Yaskawa INFORM job: DEMO_ROOF_SIDE_0625_3PAINT_42.JBI

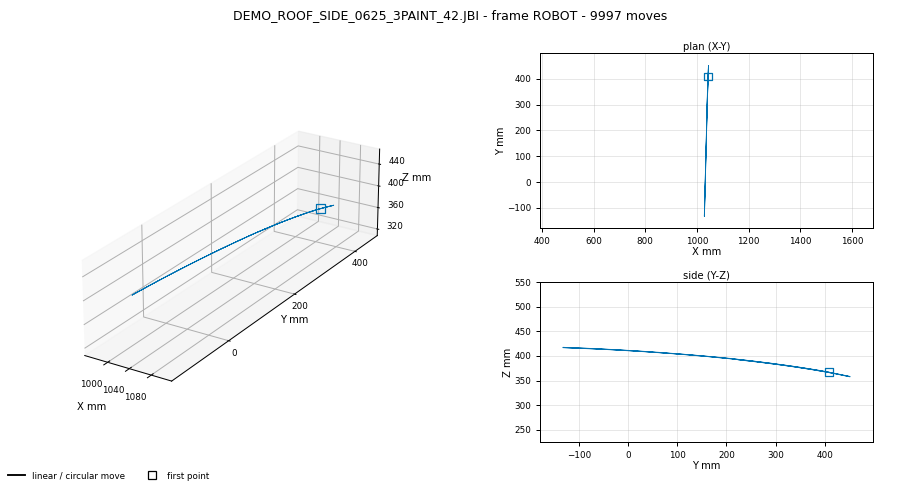
[picture p0: tool path of DEMO_ROOF_SIDE_0625_3PAINT_42.JBI in frame ROBOT, 9997 of 9997 moves have a stored position in this frame; points joined in program order, loops and branches not executed]
/JOB
//NAME DEMO_ROOF_SIDE_0625_3PAINT42
//POS
///NPOS 9997,0,0,0,0,0
///TOOL 0
///USER 0
///POSTYPE ROBOT
///RECTAN
///RCONF 1,0,0,0,0,0,0,0,0,0,0,0,0,0,0,0,0,0,0,0,0,0,0,0
C00000=1043.690,408.820,367.048,174.408,43.868,158.704
C00001=1043.680,408.575,367.094,174.398,43.862,158.701
C00002=1043.671,408.330,367.139,174.389,43.855,158.699
C00003=1043.661,408.085,367.184,174.379,43.848,158.696
C00004=1043.651,407.839,367.230,174.370,43.842,158.694
C00005=1043.642,407.593,367.275,174.361,43.835,158.691
C00006=1043.632,407.347,367.320,174.352,43.829,158.689
C00007=1043.623,407.101,367.365,174.342,43.822,158.686
C00008=1043.613,406.855,367.411,174.333,43.816,158.684
C00009=1043.603,406.610,367.456,174.325,43.809,158.681
C00010=1043.594,406.364,367.501,174.315,43.802,158.679
C00011=1043.586,406.155,367.540,174.308,43.797,158.677
C00012=1043.578,405.946,367.578,174.300,43.791,158.674
C00013=1043.570,405.736,367.616,174.292,43.786,158.672
C00014=1043.561,405.527,367.655,174.284,43.780,158.670
C00015=1043.554,405.317,367.693,174.277,43.775,158.668
C00016=1043.545,405.108,367.732,174.269,43.770,158.666
C00017=1043.537,404.898,367.770,174.261,43.764,158.664
C00018=1043.530,404.689,367.808,174.254,43.759,158.662
C00019=1043.520,404.444,367.853,174.244,43.753,158.660
C00020=1043.511,404.197,367.898,174.235,43.746,158.657
C00021=1043.502,403.952,367.942,174.226,43.740,158.655
C00022=1043.492,403.706,367.987,174.218,43.733,158.652
C00023=1043.483,403.460,368.032,174.209,43.727,158.650
C00024=1043.474,403.214,368.077,174.200,43.721,158.648
C00025=1043.464,402.968,368.121,174.191,43.715,158.645
C00026=1043.454,402.723,368.166,174.183,43.708,158.643
C00027=1043.445,402.477,368.210,174.174,43.702,158.640
C00028=1043.436,402.231,368.255,174.164,43.696,158.638
C00029=1043.427,401.985,368.299,174.156,43.690,158.636
C00030=1043.417,401.740,368.344,174.147,43.684,158.634
C00031=1043.408,401.494,368.388,174.138,43.678,158.631
C00032=1043.399,401.248,368.432,174.130,43.671,158.629
C00033=1043.390,401.002,368.476,174.121,43.666,158.627
C00034=1043.380,400.757,368.521,174.112,43.660,158.624
C00035=1043.371,400.511,368.565,174.104,43.653,158.622
C00036=1043.362,400.264,368.609,174.096,43.648,158.620
C00037=1043.353,400.019,368.653,174.086,43.641,158.617
C00038=1043.344,399.773,368.697,174.079,43.635,158.615
C00039=1043.334,399.527,368.741,174.070,43.630,158.613
C00040=1043.325,399.281,368.785,174.062,43.623,158.611
C00041=1043.315,399.035,368.829,174.053,43.618,158.609
C00042=1043.306,398.789,368.873,174.045,43.612,158.606
C00043=1043.297,398.544,368.917,174.036,43.606,158.604
C00044=1043.288,398.297,368.960,174.028,43.600,158.602
C00045=1043.279,398.051,369.004,174.019,43.594,158.600
C00046=1043.270,397.805,369.048,174.012,43.588,158.598
C00047=1043.261,397.560,369.092,174.003,43.583,158.595
C00048=1043.252,397.313,369.135,173.995,43.577,158.593
C00049=1043.243,397.068,369.179,173.986,43.571,158.591
C00050=1043.234,396.822,369.223,173.978,43.565,158.589
C00051=1043.225,396.575,369.266,173.970,43.559,158.587
C00052=1043.216,396.329,369.310,173.962,43.554,158.584
C00053=1043.206,396.084,369.353,173.953,43.548,158.582
C00054=1043.198,395.838,369.396,173.945,43.542,158.580
C00055=1043.188,395.592,369.440,173.937,43.536,158.578
C00056=1043.180,395.346,369.483,173.929,43.531,158.576
C00057=1043.171,395.100,369.526,173.921,43.525,158.574
C00058=1043.162,394.854,369.570,173.913,43.519,158.572
C00059=1043.153,394.608,369.613,173.905,43.514,158.570
C00060=1043.144,394.362,369.656,173.897,43.508,158.568
C00061=1043.135,394.116,369.700,173.889,43.502,158.565
C00062=1043.126,393.870,369.742,173.880,43.497,158.563
C00063=1043.117,393.624,369.785,173.873,43.491,158.561
C00064=1043.109,393.378,369.828,173.865,43.486,158.559
C00065=1043.100,393.131,369.872,173.856,43.480,158.557
C00066=1043.090,392.886,369.914,173.849,43.475,158.555
C00067=1043.082,392.639,369.957,173.841,43.469,158.553
C00068=1043.073,392.393,370.000,173.833,43.464,158.551
C00069=1043.064,392.148,370.043,173.825,43.458,158.549
C00070=1043.056,391.902,370.086,173.817,43.453,158.547
C00071=1043.041,391.502,370.156,173.805,43.444,158.544
C00072=1043.027,391.102,370.225,173.792,43.435,158.540
C00073=1043.012,390.702,370.294,173.780,43.426,158.537
C00074=1042.998,390.303,370.363,173.767,43.418,158.534
C00075=1042.989,390.057,370.406,173.759,43.413,158.532
C00076=1042.981,389.811,370.449,173.752,43.407,158.530
C00077=1042.972,389.565,370.491,173.744,43.402,158.528
C00078=1042.963,389.319,370.534,173.737,43.397,158.526
C00079=1042.954,389.073,370.576,173.729,43.391,158.524
C00080=1042.946,388.826,370.619,173.722,43.386,158.522
C00081=1042.937,388.580,370.661,173.713,43.381,158.520
C00082=1042.929,388.334,370.703,173.706,43.376,158.519
C00083=1042.919,388.088,370.746,173.698,43.371,158.517
C00084=1042.910,387.842,370.787,173.691,43.365,158.515
C00085=1042.902,387.595,370.830,173.683,43.360,158.513
C00086=1042.893,387.349,370.872,173.676,43.355,158.511
C00087=1042.884,387.103,370.914,173.669,43.350,158.509
C00088=1042.876,386.856,370.956,173.661,43.345,158.507
C00089=1042.867,386.610,370.998,173.654,43.340,158.505
C00090=1042.859,386.364,371.039,173.646,43.334,158.503
C00091=1042.849,386.118,371.082,173.639,43.330,158.502
C00092=1042.841,385.872,371.124,173.632,43.324,158.500
C00093=1042.832,385.625,371.166,173.624,43.319,158.498
C00094=1042.823,385.379,371.207,173.617,43.315,158.496
C00095=1042.815,385.133,371.249,173.609,43.309,158.494
C00096=1042.807,384.887,371.291,173.602,43.304,158.492
C00097=1042.798,384.640,371.333,173.595,43.300,158.490
C00098=1042.789,384.394,371.375,173.588,43.295,158.489
C00099=1042.781,384.148,371.416,173.580,43.289,158.487
C00100=1042.772,383.902,371.458,173.573,43.284,158.485
C00101=1042.763,383.655,371.500,173.566,43.280,158.483
C00102=1042.755,383.409,371.541,173.558,43.275,158.481
C00103=1042.746,383.163,371.582,173.551,43.270,158.480
C00104=1042.738,382.916,371.625,173.545,43.265,158.478
C00105=1042.730,382.670,371.666,173.538,43.260,158.476
C00106=1042.721,382.423,371.707,173.530,43.255,158.474
C00107=1042.712,382.177,371.749,173.523,43.250,158.472
C00108=1042.705,381.931,371.791,173.516,43.245,158.471
C00109=1042.696,381.684,371.832,173.508,43.241,158.469
C00110=1042.688,381.438,371.873,173.501,43.236,158.467
C00111=1042.679,381.192,371.915,173.495,43.231,158.465
C00112=1042.672,380.945,371.956,173.488,43.226,158.464
C00113=1042.663,380.699,371.998,173.480,43.221,158.462
C00114=1042.655,380.453,372.038,173.473,43.217,158.460
C00115=1042.646,380.206,372.080,173.466,43.212,158.458
C00116=1042.638,379.960,372.121,173.460,43.207,158.457
C00117=1042.629,379.713,372.163,173.453,43.202,158.455
C00118=1042.621,379.467,372.203,173.446,43.198,158.453
C00119=1042.613,379.221,372.244,173.438,43.193,158.451
C00120=1042.604,378.974,372.286,173.432,43.188,158.450
C00121=1042.596,378.728,372.326,173.425,43.183,158.448
C00122=1042.588,378.481,372.367,173.418,43.178,158.446
C00123=1042.580,378.235,372.408,173.411,43.174,158.445
C00124=1042.571,377.988,372.449,173.405,43.170,158.443
C00125=1042.563,377.742,372.490,173.398,43.165,158.441
C00126=1042.555,377.495,372.530,173.391,43.160,158.440
C00127=1042.542,377.130,372.591,173.380,43.154,158.437
C00128=1042.530,376.764,372.651,173.370,43.147,158.435
C00129=1042.518,376.398,372.712,173.360,43.140,158.432
C00130=1042.505,376.032,372.772,173.351,43.133,158.430
C00131=1042.497,375.786,372.813,173.344,43.128,158.428
C00132=1042.489,375.539,372.854,173.337,43.124,158.427
C00133=1042.481,375.292,372.894,173.331,43.120,158.425
C00134=1042.472,375.046,372.934,173.324,43.115,158.423
C00135=1042.464,374.799,372.974,173.317,43.111,158.422
C00136=1042.456,374.552,373.015,173.311,43.106,158.420
C00137=1042.448,374.306,373.056,173.304,43.102,158.419
C00138=1042.440,374.059,373.096,173.298,43.098,158.417
C00139=1042.432,373.813,373.137,173.291,43.093,158.416
C00140=1042.424,373.567,373.177,173.284,43.089,158.414
C00141=1042.415,373.319,373.217,173.278,43.084,158.412
C00142=1042.407,373.073,373.257,173.271,43.080,158.411
C00143=1042.399,372.827,373.298,173.265,43.076,158.409
C00144=1042.391,372.580,373.338,173.258,43.071,158.408
C00145=1042.383,372.334,373.379,173.252,43.067,158.406
C00146=1042.375,372.087,373.419,173.245,43.062,158.404
C00147=1042.367,371.840,373.459,173.239,43.058,158.403
C00148=1042.359,371.594,373.499,173.232,43.054,158.401
C00149=1042.351,371.348,373.539,173.226,43.050,158.400
C00150=1042.343,371.101,373.579,173.219,43.045,158.398
C00151=1042.335,370.854,373.619,173.213,43.041,158.397
C00152=1042.327,370.608,373.660,173.206,43.037,158.395
C00153=1042.319,370.361,373.699,173.200,43.032,158.394
C00154=1042.311,370.114,373.739,173.193,43.028,158.392
C00155=1042.303,369.867,373.778,173.188,43.024,158.391
C00156=1042.295,369.621,373.818,173.181,43.020,158.389
C00157=1042.286,369.375,373.858,173.175,43.016,158.388
C00158=1042.278,369.128,373.898,173.169,43.011,158.386
C00159=1042.270,368.881,373.937,173.162,43.007,158.385
C00160=1042.262,368.634,373.977,173.156,43.003,158.383
C00161=1042.254,368.388,374.017,173.149,42.999,158.382
C00162=1042.246,368.141,374.057,173.144,42.995,158.380
C00163=1042.238,367.894,374.096,173.137,42.991,158.379
C00164=1042.230,367.647,374.136,173.131,42.987,158.377
C00165=1042.221,367.401,374.175,173.125,42.983,158.376
C00166=1042.214,367.154,374.215,173.118,42.978,158.374
C00167=1042.206,366.907,374.253,173.112,42.974,158.373
C00168=1042.198,366.660,374.293,173.107,42.970,158.371
C00169=1042.190,366.414,374.333,173.100,42.966,158.370
C00170=1042.182,366.167,374.372,173.094,42.962,158.368
C00171=1042.174,365.920,374.412,173.088,42.958,158.367
C00172=1042.166,365.673,374.452,173.081,42.954,158.366
C00173=1042.158,365.427,374.490,173.076,42.950,158.364
C00174=1042.151,365.180,374.530,173.070,42.946,158.363
C00175=1042.142,364.933,374.569,173.063,42.942,158.361
C00176=1042.135,364.686,374.608,173.057,42.938,158.360
C00177=1042.127,364.440,374.647,173.051,42.934,158.358
C00178=1042.119,364.193,374.687,173.045,42.930,158.357
C00179=1042.111,363.946,374.726,173.039,42.926,158.356
C00180=1042.104,363.699,374.765,173.033,42.922,158.354
C00181=1042.096,363.452,374.804,173.027,42.918,158.353
C00182=1042.088,363.205,374.844,173.021,42.914,158.351
C00183=1042.077,362.859,374.898,173.012,42.909,158.349
C00184=1042.066,362.513,374.953,173.004,42.904,158.348
C00185=1042.056,362.168,375.008,172.997,42.898,158.346
C00186=1042.045,361.821,375.062,172.988,42.893,158.344
C00187=1042.037,361.574,375.101,172.981,42.889,158.342
C00188=1042.028,361.327,375.140,172.976,42.885,158.341
C00189=1042.021,361.081,375.178,172.970,42.881,158.340
C00190=1042.013,360.833,375.218,172.964,42.877,158.338
C00191=1042.006,360.587,375.256,172.959,42.873,158.337
C00192=1041.997,360.340,375.295,172.952,42.870,158.335
C00193=1041.989,360.093,375.334,172.946,42.866,158.334
C00194=1041.982,359.847,375.372,172.941,42.862,158.333
C00195=1041.974,359.599,375.411,172.935,42.859,158.332
C00196=1041.967,359.353,375.450,172.929,42.855,158.330
C00197=1041.959,359.105,375.488,172.923,42.851,158.329
C00198=1041.951,358.859,375.526,172.917,42.847,158.328
C00199=1041.943,358.612,375.565,172.911,42.843,158.326
C00200=1041.935,358.365,375.603,172.906,42.840,158.325
C00201=1041.927,358.118,375.642,172.900,42.836,158.324
C00202=1041.920,357.871,375.680,172.895,42.833,158.322
C00203=1041.912,357.624,375.719,172.889,42.829,158.321
C00204=1041.905,357.377,375.758,172.883,42.825,158.320
C00205=1041.897,357.131,375.796,172.877,42.822,158.318
C00206=1041.889,356.884,375.834,172.871,42.818,158.317
C00207=1041.882,356.636,375.872,172.866,42.814,158.316
C00208=1041.874,356.389,375.911,172.860,42.810,158.314
C00209=1041.866,356.143,375.949,172.854,42.807,158.313
C00210=1041.859,355.896,375.987,172.849,42.803,158.312
C00211=1041.851,355.648,376.025,172.843,42.800,158.311
C00212=1041.843,355.402,376.063,172.838,42.796,158.309
C00213=1041.835,355.155,376.102,172.832,42.793,158.308
C00214=1041.828,354.908,376.139,172.827,42.789,158.307
C00215=1041.820,354.661,376.178,172.821,42.786,158.306
C00216=1041.812,354.413,376.215,172.816,42.782,158.305
C00217=1041.804,354.167,376.253,172.810,42.779,158.303
C00218=1041.797,353.920,376.291,172.804,42.775,158.302
C00219=1041.789,353.673,376.329,172.799,42.771,158.301
C00220=1041.781,353.425,376.367,172.792,42.768,158.299
C00221=1041.774,353.179,376.405,172.787,42.765,158.298
C00222=1041.767,352.932,376.443,172.781,42.761,158.297
C00223=1041.759,352.685,376.481,172.776,42.758,158.296
C00224=1041.751,352.437,376.519,172.771,42.754,158.295
C00225=1041.744,352.191,376.557,172.766,42.751,158.293
C00226=1041.736,351.944,376.594,172.760,42.747,158.292
C00227=1041.729,351.697,376.632,172.755,42.744,158.291
C00228=1041.722,351.450,376.670,172.749,42.740,158.290
C00229=1041.713,351.203,376.707,172.744,42.737,158.288
C00230=1041.706,350.955,376.745,172.738,42.733,158.287
C00231=1041.699,350.708,376.783,172.733,42.730,158.286
C00232=1041.691,350.462,376.821,172.727,42.726,158.285
C00233=1041.684,350.215,376.858,172.722,42.723,158.284
C00234=1041.677,349.968,376.896,172.717,42.720,158.283
C00235=1041.669,349.720,376.933,172.711,42.717,158.281
C00236=1041.661,349.473,376.971,172.706,42.713,158.280
C00237=1041.653,349.226,377.008,172.700,42.710,158.279
C00238=1041.646,348.979,377.046,172.695,42.706,158.278
C00239=1041.636,348.639,377.097,172.688,42.702,158.276
C00240=1041.625,348.299,377.148,172.681,42.697,158.275
C00241=1041.615,347.958,377.200,172.673,42.693,158.273
C00242=1041.604,347.618,377.251,172.666,42.688,158.271
C00243=1041.596,347.371,377.288,172.660,42.685,158.270
C00244=1041.589,347.124,377.326,172.655,42.682,158.269
C00245=1041.582,346.877,377.363,172.650,42.679,158.268
C00246=1041.574,346.630,377.400,172.644,42.675,158.267
C00247=1041.567,346.383,377.438,172.640,42.672,158.266
C00248=1041.560,346.135,377.474,172.634,42.669,158.264
C00249=1041.552,345.888,377.511,172.629,42.666,158.263
C00250=1041.545,345.641,377.549,172.624,42.662,158.262
C00251=1041.537,345.394,377.586,172.618,42.659,158.261
C00252=1041.530,345.146,377.623,172.613,42.656,158.260
C00253=1041.522,344.899,377.660,172.609,42.653,158.259
C00254=1041.515,344.653,377.697,172.603,42.649,158.258
C00255=1041.508,344.405,377.734,172.598,42.646,158.257
C00256=1041.500,344.159,377.771,172.592,42.643,158.255
C00257=1041.493,343.911,377.808,172.587,42.640,158.254
C00258=1041.485,343.664,377.844,172.583,42.637,158.253
C00259=1041.478,343.417,377.882,172.577,42.634,158.252
C00260=1041.471,343.169,377.919,172.572,42.631,158.251
C00261=1041.463,342.922,377.956,172.567,42.628,158.250
C00262=1041.457,342.675,377.992,172.562,42.624,158.249
C00263=1041.449,342.428,378.029,172.557,42.621,158.248
C00264=1041.442,342.181,378.066,172.552,42.618,158.247
C00265=1041.434,341.934,378.103,172.546,42.615,158.245
C00266=1041.427,341.686,378.139,172.542,42.612,158.244
C00267=1041.419,341.439,378.176,172.537,42.609,158.243
C00268=1041.412,341.193,378.212,172.532,42.606,158.242
C00269=1041.404,340.945,378.248,172.526,42.603,158.241
C00270=1041.397,340.697,378.285,172.522,42.599,158.240
C00271=1041.389,340.450,378.322,172.517,42.596,158.239
C00272=1041.381,340.203,378.358,172.511,42.594,158.238
C00273=1041.375,339.956,378.395,172.506,42.591,158.237
C00274=1041.367,339.709,378.431,172.502,42.588,158.236
C00275=1041.360,339.461,378.467,172.496,42.585,158.235
C00276=1041.352,339.214,378.504,172.491,42.582,158.234
C00277=1041.345,338.967,378.541,172.487,42.579,158.233
C00278=1041.338,338.720,378.577,172.482,42.576,158.232
C00279=1041.330,338.472,378.613,172.476,42.573,158.231
C00280=1041.324,338.225,378.650,172.472,42.570,158.230
C00281=1041.316,337.978,378.686,172.467,42.567,158.229
C00282=1041.308,337.730,378.722,172.462,42.564,158.228
C00283=1041.301,337.484,378.758,172.457,42.561,158.227
C00284=1041.294,337.236,378.795,172.452,42.558,158.225
C00285=1041.287,336.988,378.831,172.447,42.555,158.224
C00286=1041.280,336.742,378.867,172.443,42.552,158.223
C00287=1041.272,336.494,378.903,172.437,42.549,158.222
C00288=1041.266,336.247,378.939,172.432,42.546,158.221
C00289=1041.258,336.000,378.976,172.428,42.543,158.220
C00290=1041.250,335.752,379.012,172.423,42.540,158.219
C00291=1041.243,335.506,379.048,172.419,42.538,158.218
C00292=1041.237,335.257,379.084,172.413,42.535,158.217
C00293=1041.230,335.010,379.120,172.408,42.532,158.216
C00294=1041.222,334.763,379.156,172.404,42.529,158.215
C00295=1041.211,334.419,379.205,172.397,42.525,158.214
C00296=1041.201,334.076,379.255,172.390,42.521,158.212
C00297=1041.191,333.732,379.305,172.384,42.517,158.211
C00298=1041.182,333.388,379.355,172.377,42.514,158.210
C00299=1041.174,333.140,379.391,172.372,42.511,158.209
C00300=1041.167,332.893,379.426,172.368,42.507,158.208
C00301=1041.159,332.646,379.463,172.363,42.505,158.207
C00302=1041.153,332.398,379.498,172.357,42.502,158.206
C00303=1041.145,332.151,379.534,172.353,42.499,158.205
C00304=1041.138,331.903,379.569,172.348,42.497,158.204
C00305=1041.131,331.656,379.605,172.344,42.494,158.203
C00306=1041.124,331.409,379.641,172.339,42.491,158.202
C00307=1041.116,331.161,379.677,172.335,42.488,158.201
C00308=1041.109,330.914,379.712,172.329,42.485,158.200
C00309=1041.102,330.667,379.748,172.325,42.483,158.199
C00310=1041.095,330.419,379.783,172.320,42.480,158.198
C00311=1041.088,330.172,379.819,172.316,42.477,158.197
C00312=1041.080,329.924,379.855,172.311,42.474,158.196
C00313=1041.073,329.677,379.890,172.307,42.472,158.195
C00314=1041.067,329.430,379.926,172.302,42.469,158.194
C00315=1041.059,329.182,379.960,172.297,42.467,158.193
C00316=1041.051,328.936,379.996,172.292,42.464,158.192
C00317=1041.045,328.688,380.031,172.288,42.461,158.192
C00318=1041.037,328.440,380.067,172.283,42.459,158.191
C00319=1041.030,328.193,380.101,172.279,42.456,158.190
C00320=1041.022,327.945,380.137,172.274,42.453,158.189
C00321=1041.015,327.698,380.172,172.270,42.451,158.188
C00322=1041.008,327.451,380.207,172.265,42.448,158.187
C00323=1041.000,327.203,380.243,172.261,42.445,158.186
C00324=1040.993,326.956,380.277,172.256,42.443,158.185
C00325=1040.986,326.709,380.313,172.251,42.440,158.184
C00326=1040.978,326.461,380.347,172.246,42.438,158.183
C00327=1040.971,326.214,380.383,172.242,42.435,158.182
C00328=1040.964,325.967,380.417,172.237,42.433,158.181
C00329=1040.956,325.718,380.453,172.233,42.430,158.181
C00330=1040.950,325.471,380.488,172.228,42.428,158.180
C00331=1040.942,325.224,380.522,172.224,42.425,158.179
C00332=1040.935,324.977,380.557,172.219,42.423,158.178
C00333=1040.928,324.728,380.592,172.215,42.420,158.177
C00334=1040.921,324.481,380.627,172.211,42.417,158.176
C00335=1040.913,324.234,380.661,172.206,42.415,158.175
C00336=1040.907,323.987,380.696,172.202,42.412,158.174
C00337=1040.898,323.739,380.731,172.197,42.410,158.173
C00338=1040.892,323.491,380.766,172.193,42.408,158.173
C00339=1040.885,323.244,380.802,172.188,42.405,158.172
C00340=1040.878,322.996,380.835,172.184,42.403,158.171
C00341=1040.871,322.749,380.871,172.180,42.400,158.170
C00342=1040.863,322.502,380.905,172.174,42.398,158.169
C00343=1040.856,322.254,380.941,172.170,42.395,158.168
C00344=1040.849,322.006,380.974,172.166,42.392,158.167
C00345=1040.842,321.759,381.010,172.161,42.390,158.166
C00346=1040.835,321.512,381.044,172.157,42.387,158.166
C00347=1040.828,321.264,381.079,172.152,42.385,158.165
C00348=1040.821,321.017,381.113,172.148,42.382,158.164
C00349=1040.814,320.769,381.148,172.144,42.380,158.163
C00350=1040.807,320.522,381.182,172.139,42.377,158.162
C00351=1040.797,320.173,381.232,172.134,42.374,158.161
C00352=1040.787,319.825,381.280,172.127,42.370,158.160
C00353=1040.777,319.476,381.329,172.121,42.367,158.158
C00354=1040.767,319.127,381.377,172.115,42.363,158.157
C00355=1040.760,318.879,381.412,172.110,42.362,158.156
C00356=1040.753,318.632,381.446,172.106,42.359,158.156
C00357=1040.746,318.384,381.481,172.102,42.357,158.155
C00358=1040.739,318.137,381.515,172.097,42.354,158.154
C00359=1040.732,317.889,381.550,172.093,42.352,158.153
C00360=1040.725,317.642,381.584,172.089,42.349,158.152
C00361=1040.718,317.394,381.619,172.085,42.347,158.151
C00362=1040.711,317.147,381.653,172.080,42.344,158.150
C00363=1040.704,316.899,381.688,172.076,42.342,158.150
C00364=1040.697,316.651,381.721,172.072,42.340,158.149
C00365=1040.691,316.405,381.756,172.068,42.337,158.148
C00366=1040.684,316.157,381.790,172.063,42.335,158.147
C00367=1040.677,315.909,381.824,172.059,42.332,158.146
C00368=1040.670,315.662,381.859,172.055,42.330,158.145
C00369=1040.663,315.414,381.893,172.052,42.328,158.145
C00370=1040.656,315.166,381.927,172.046,42.326,158.144
C00371=1040.649,314.919,381.962,172.042,42.323,158.143
C00372=1040.643,314.672,381.996,172.038,42.320,158.142
C00373=1040.636,314.424,382.030,172.034,42.318,158.141
C00374=1040.629,314.176,382.064,172.030,42.316,158.141
C00375=1040.622,313.929,382.099,172.026,42.314,158.140
C00376=1040.615,313.681,382.133,172.022,42.311,158.139
C00377=1040.609,313.434,382.167,172.018,42.309,158.138
C00378=1040.601,313.187,382.200,172.014,42.307,158.137
C00379=1040.595,312.939,382.235,172.010,42.304,158.137
C00380=1040.588,312.691,382.269,172.005,42.302,158.136
C00381=1040.582,312.444,382.303,172.001,42.300,158.135
C00382=1040.574,312.197,382.337,171.997,42.297,158.134
C00383=1040.567,311.949,382.371,171.993,42.295,158.133
C00384=1040.560,311.701,382.404,171.989,42.293,158.133
C00385=1040.553,311.453,382.438,171.984,42.290,158.132
C00386=1040.547,311.206,382.471,171.980,42.288,158.131
C00387=1040.539,310.958,382.505,171.976,42.286,158.130
C00388=1040.532,310.711,382.539,171.972,42.284,158.129
C00389=1040.524,310.463,382.572,171.968,42.282,158.129
C00390=1040.517,310.216,382.606,171.963,42.280,158.128
C00391=1040.511,309.968,382.639,171.960,42.278,158.127
C00392=1040.504,309.720,382.673,171.956,42.276,158.126
C00393=1040.496,309.473,382.706,171.952,42.273,158.126
C00394=1040.489,309.225,382.740,171.947,42.271,158.125
C00395=1040.483,308.978,382.773,171.943,42.269,158.124
C00396=1040.476,308.730,382.807,171.939,42.267,158.123
C00397=1040.468,308.482,382.840,171.935,42.265,158.123
C00398=1040.460,308.235,382.874,171.931,42.262,158.122
C00399=1040.454,307.987,382.907,171.928,42.260,158.121
C00400=1040.447,307.740,382.940,171.923,42.259,158.120
C00401=1040.440,307.491,382.974,171.919,42.256,158.120
C00402=1040.433,307.244,383.007,171.915,42.254,158.119
C00403=1040.426,306.997,383.040,171.911,42.252,158.118
C00404=1040.419,306.749,383.073,171.907,42.250,158.117
C00405=1040.412,306.502,383.107,171.903,42.248,158.117
C00406=1040.405,306.253,383.140,171.899,42.246,158.116
C00407=1040.396,305.910,383.187,171.893,42.243,158.115
C00408=1040.386,305.566,383.233,171.888,42.240,158.114
C00409=1040.377,305.222,383.279,171.883,42.237,158.113
C00410=1040.367,304.878,383.325,171.877,42.234,158.112
C00411=1040.359,304.631,383.358,171.873,42.232,158.111
C00412=1040.352,304.383,383.391,171.869,42.230,158.110
C00413=1040.346,304.136,383.424,171.865,42.227,158.110
C00414=1040.339,303.887,383.458,171.861,42.225,158.109
C00415=1040.332,303.639,383.491,171.857,42.223,158.108
C00416=1040.326,303.392,383.524,171.854,42.222,158.107
C00417=1040.318,303.144,383.557,171.850,42.219,158.107
C00418=1040.311,302.897,383.590,171.846,42.217,158.106
C00419=1040.304,302.649,383.623,171.842,42.215,158.105
C00420=1040.298,302.401,383.656,171.838,42.213,158.105
C00421=1040.291,302.154,383.690,171.834,42.211,158.104
C00422=1040.284,301.906,383.722,171.830,42.209,158.103
C00423=1040.277,301.658,383.755,171.826,42.207,158.102
C00424=1040.271,301.411,383.788,171.823,42.205,158.102
C00425=1040.264,301.164,383.821,171.819,42.203,158.101
C00426=1040.257,300.915,383.854,171.815,42.201,158.100
C00427=1040.250,300.668,383.886,171.810,42.199,158.100
C00428=1040.243,300.420,383.920,171.806,42.196,158.099
C00429=1040.237,300.173,383.953,171.802,42.194,158.098
C00430=1040.230,299.924,383.986,171.799,42.192,158.097
C00431=1040.223,299.677,384.018,171.795,42.190,158.097
C00432=1040.216,299.430,384.051,171.791,42.188,158.096
C00433=1040.210,299.181,384.084,171.788,42.186,158.095
C00434=1040.203,298.934,384.117,171.784,42.184,158.095
C00435=1040.197,298.686,384.150,171.781,42.182,158.094
C00436=1040.189,298.439,384.183,171.777,42.180,158.093
C00437=1040.183,298.191,384.216,171.773,42.178,158.092
C00438=1040.176,297.944,384.248,171.769,42.176,158.092
C00439=1040.170,297.695,384.281,171.765,42.174,158.091
C00440=1040.163,297.448,384.314,171.761,42.172,158.090
C00441=1040.156,297.200,384.346,171.758,42.170,158.090
C00442=1040.149,296.952,384.379,171.754,42.168,158.089
C00443=1040.143,296.704,384.412,171.750,42.166,158.088
C00444=1040.136,296.457,384.444,171.746,42.164,158.088
C00445=1040.129,296.209,384.477,171.742,42.162,158.087
C00446=1040.123,295.961,384.510,171.739,42.160,158.086
C00447=1040.117,295.714,384.543,171.735,42.158,158.085
C00448=1040.109,295.466,384.575,171.731,42.156,158.085
C00449=1040.103,295.218,384.607,171.727,42.154,158.084
C00450=1040.096,294.970,384.640,171.723,42.152,158.083
C00451=1040.090,294.723,384.672,171.721,42.150,158.083
C00452=1040.082,294.475,384.705,171.717,42.148,158.082
C00453=1040.076,294.227,384.738,171.713,42.146,158.081
C00454=1040.069,293.979,384.769,171.709,42.144,158.081
C00455=1040.063,293.732,384.802,171.705,42.143,158.080
C00456=1040.055,293.484,384.834,171.702,42.141,158.079
C00457=1040.049,293.236,384.867,171.698,42.139,158.079
C00458=1040.042,292.988,384.898,171.694,42.137,158.078
C00459=1040.034,292.740,384.931,171.690,42.135,158.077
C00460=1040.028,292.492,384.963,171.687,42.134,158.077
C00461=1040.021,292.245,384.995,171.683,42.132,158.076
C00462=1040.014,291.997,385.027,171.679,42.130,158.075
C00463=1040.006,291.669,385.069,171.675,42.127,158.075
C00464=1039.996,291.342,385.112,171.670,42.125,158.074
C00465=1039.987,291.015,385.155,171.665,42.122,158.073
C00466=1039.979,290.687,385.197,171.660,42.120,158.072
C00467=1039.972,290.440,385.229,171.656,42.118,158.071
C00468=1039.966,290.192,385.261,171.653,42.116,158.071
C00469=1039.959,289.944,385.293,171.650,42.114,158.070
C00470=1039.951,289.696,385.325,171.646,42.112,158.069
C00471=1039.944,289.448,385.357,171.642,42.110,158.069
C00472=1039.938,289.200,385.389,171.639,42.109,158.068
C00473=1039.931,288.953,385.421,171.635,42.107,158.068
C00474=1039.924,288.705,385.453,171.631,42.105,158.067
C00475=1039.918,288.457,385.484,171.627,42.104,158.066
C00476=1039.911,288.209,385.517,171.625,42.101,158.066
C00477=1039.904,287.961,385.549,171.621,42.099,158.065
C00478=1039.897,287.714,385.581,171.617,42.098,158.064
C00479=1039.890,287.466,385.612,171.613,42.096,158.064
C00480=1039.884,287.218,385.644,171.610,42.094,158.063
C00481=1039.878,286.970,385.676,171.606,42.093,158.062
C00482=1039.871,286.722,385.708,171.603,42.091,158.062
C00483=1039.864,286.475,385.739,171.599,42.089,158.061
C00484=1039.857,286.226,385.771,171.596,42.087,158.061
C00485=1039.850,285.978,385.802,171.592,42.085,158.060
C00486=1039.843,285.731,385.835,171.588,42.084,158.059
C00487=1039.836,285.483,385.866,171.585,42.082,158.059
C00488=1039.829,285.235,385.897,171.582,42.080,158.058
C00489=1039.823,284.987,385.929,171.578,42.078,158.058
C00490=1039.816,284.739,385.960,171.575,42.077,158.057
C00491=1039.809,284.491,385.992,171.571,42.075,158.056
C00492=1039.802,284.243,386.023,171.567,42.074,158.056
C00493=1039.796,283.995,386.055,171.564,42.071,158.055
C00494=1039.789,283.747,386.086,171.561,42.070,158.055
C00495=1039.782,283.500,386.117,171.557,42.068,158.054
C00496=1039.775,283.252,386.150,171.553,42.066,158.053
C00497=1039.768,283.004,386.181,171.551,42.065,158.053
C00498=1039.761,282.756,386.213,171.547,42.063,158.052
C00499=1039.754,282.508,386.244,171.543,42.061,158.051
C00500=1039.748,282.260,386.276,171.540,42.059,158.051
C00501=1039.741,282.012,386.307,171.537,42.058,158.050
C00502=1039.735,281.764,386.338,171.533,42.056,158.050
C00503=1039.728,281.516,386.369,171.530,42.054,158.049
C00504=1039.722,281.268,386.400,171.526,42.053,158.049
C00505=1039.715,281.021,386.432,171.523,42.051,158.048
C00506=1039.708,280.773,386.463,171.520,42.049,158.047
C00507=1039.702,280.525,386.495,171.516,42.047,158.047
C00508=1039.695,280.277,386.526,171.512,42.046,158.046
C00509=1039.688,280.029,386.557,171.509,42.044,158.045
C00510=1039.681,279.781,386.589,171.506,42.042,158.045
C00511=1039.675,279.533,386.620,171.502,42.040,158.044
C00512=1039.668,279.285,386.651,171.499,42.039,158.044
C00513=1039.662,279.037,386.682,171.496,42.037,158.043
C00514=1039.655,278.789,386.714,171.492,42.036,158.043
C00515=1039.647,278.541,386.745,171.488,42.034,158.042
C00516=1039.641,278.293,386.775,171.486,42.032,158.041
C00517=1039.634,278.045,386.807,171.482,42.031,158.041
C00518=1039.628,277.798,386.838,171.478,42.029,158.040
C00519=1039.618,277.482,386.877,171.474,42.027,158.039
C00520=1039.610,277.166,386.917,171.470,42.025,158.039
C00521=1039.602,276.851,386.957,171.466,42.023,158.038
C00522=1039.594,276.535,386.995,171.462,42.020,158.037
C00523=1039.586,276.287,387.026,171.458,42.019,158.037
C00524=1039.580,276.040,387.058,171.455,42.017,158.036
C00525=1039.573,275.791,387.088,171.451,42.016,158.036
C00526=1039.566,275.544,387.119,171.448,42.014,158.035
C00527=1039.560,275.296,387.150,171.445,42.012,158.034
C00528=1039.553,275.048,387.181,171.441,42.011,158.034
C00529=1039.547,274.799,387.212,171.438,42.009,158.033
C00530=1039.539,274.552,387.243,171.435,42.007,158.033
C00531=1039.533,274.303,387.273,171.432,42.006,158.032
C00532=1039.527,274.056,387.304,171.428,42.004,158.032
C00533=1039.520,273.808,387.335,171.425,42.003,158.031
C00534=1039.513,273.560,387.366,171.422,42.001,158.030
C00535=1039.506,273.311,387.397,171.419,42.000,158.030
C00536=1039.499,273.064,387.428,171.415,41.998,158.029
C00537=1039.493,272.815,387.458,171.412,41.996,158.029
C00538=1039.486,272.568,387.489,171.409,41.995,158.028
C00539=1039.479,272.320,387.519,171.405,41.993,158.028
C00540=1039.473,272.071,387.550,171.402,41.991,158.027
C00541=1039.465,271.824,387.581,171.399,41.990,158.027
C00542=1039.460,271.576,387.611,171.396,41.988,158.026
C00543=1039.453,271.327,387.642,171.392,41.987,158.025
C00544=1039.446,271.080,387.673,171.389,41.985,158.025
C00545=1039.439,270.831,387.704,171.386,41.983,158.024
C00546=1039.433,270.584,387.733,171.382,41.982,158.024
C00547=1039.426,270.335,387.764,171.379,41.980,158.023
C00548=1039.419,270.087,387.795,171.376,41.979,158.023
C00549=1039.412,269.839,387.826,171.373,41.977,158.022
C00550=1039.406,269.591,387.855,171.370,41.976,158.022
C00551=1039.399,269.343,387.886,171.366,41.974,158.021
C00552=1039.392,269.095,387.916,171.363,41.973,158.020
C00553=1039.386,268.847,387.948,171.360,41.971,158.020
C00554=1039.379,268.599,387.977,171.356,41.970,158.019
C00555=1039.373,268.351,388.008,171.354,41.968,158.019
C00556=1039.365,268.103,388.038,171.350,41.967,158.018
C00557=1039.359,267.855,388.068,171.348,41.965,158.018
C00558=1039.352,267.606,388.099,171.344,41.964,158.017
C00559=1039.345,267.358,388.129,171.340,41.962,158.017
C00560=1039.339,267.110,388.159,171.338,41.960,158.016
C00561=1039.332,266.862,388.189,171.334,41.959,158.016
C00562=1039.325,266.614,388.219,171.332,41.957,158.015
C00563=1039.319,266.366,388.250,171.328,41.956,158.015
C00564=1039.312,266.118,388.280,171.325,41.954,158.014
C00565=1039.305,265.870,388.310,171.322,41.953,158.014
C00566=1039.299,265.622,388.340,171.319,41.951,158.013
C00567=1039.292,265.374,388.371,171.316,41.950,158.013
C00568=1039.285,265.126,388.401,171.312,41.948,158.012
C00569=1039.279,264.878,388.431,171.309,41.947,158.012
C00570=1039.272,264.630,388.461,171.306,41.945,158.011
C00571=1039.265,264.382,388.491,171.303,41.944,158.011
C00572=1039.259,264.133,388.522,171.300,41.943,158.010
C00573=1039.252,263.885,388.552,171.297,41.941,158.009
C00574=1039.245,263.638,388.581,171.293,41.940,158.009
C00575=1039.238,263.326,388.619,171.290,41.938,158.008
C00576=1039.229,263.016,388.657,171.286,41.936,158.008
C00577=1039.220,262.704,388.694,171.282,41.933,158.007
C00578=1039.212,262.393,388.732,171.278,41.931,158.006
C00579=1039.205,262.146,388.762,171.275,41.930,158.006
C00580=1039.198,261.897,388.792,171.272,41.929,158.005
C00581=1039.192,261.650,388.822,171.269,41.927,158.005
C00582=1039.185,261.401,388.851,171.266,41.926,158.004
C00583=1039.178,261.153,388.881,171.263,41.925,158.004
C00584=1039.171,260.905,388.911,171.260,41.923,158.003
C00585=1039.164,260.657,388.940,171.256,41.922,158.003
C00586=1039.158,260.409,388.970,171.254,41.920,158.002
C00587=1039.151,260.160,389.000,171.250,41.919,158.002
C00588=1039.144,259.912,389.030,171.248,41.917,158.001
C00589=1039.137,259.664,389.059,171.244,41.916,158.001
C00590=1039.130,259.416,389.089,171.242,41.915,158.000
C00591=1039.124,259.168,389.119,171.238,41.914,158.000
C00592=1039.116,258.920,389.147,171.235,41.912,157.999
C00593=1039.110,258.672,389.177,171.232,41.911,157.999
C00594=1039.103,258.423,389.207,171.229,41.909,157.998
C00595=1039.096,258.176,389.236,171.226,41.908,157.998
C00596=1039.089,257.927,389.266,171.223,41.907,157.997
C00597=1039.083,257.679,389.296,171.220,41.905,157.997
C00598=1039.076,257.431,389.325,171.217,41.904,157.996
C00599=1039.069,257.183,389.355,171.214,41.902,157.996
C00600=1039.063,256.934,389.384,171.211,41.901,157.995
C00601=1039.056,256.687,389.414,171.208,41.900,157.995
C00602=1039.049,256.438,389.443,171.205,41.898,157.994
C00603=1039.042,256.191,389.472,171.202,41.897,157.994
C00604=1039.035,255.942,389.502,171.199,41.895,157.993
C00605=1039.029,255.694,389.531,171.196,41.894,157.993
C00606=1039.022,255.445,389.561,171.193,41.892,157.992
C00607=1039.015,255.197,389.590,171.190,41.891,157.992
C00608=1039.008,254.949,389.620,171.187,41.890,157.992
C00609=1039.002,254.701,389.649,171.184,41.888,157.991
C00610=1038.995,254.452,389.679,171.182,41.887,157.991
C00611=1038.989,254.205,389.708,171.178,41.885,157.990
C00612=1038.982,253.957,389.737,171.175,41.884,157.990
C00613=1038.975,253.708,389.766,171.172,41.883,157.989
C00614=1038.968,253.460,389.795,171.169,41.882,157.989
C00615=1038.961,253.212,389.825,171.166,41.880,157.988
C00616=1038.955,252.964,389.854,171.163,41.879,157.988
C00617=1038.949,252.715,389.883,171.161,41.877,157.987
C00618=1038.942,252.467,389.914,171.157,41.876,157.987
C00619=1038.935,252.219,389.943,171.155,41.875,157.986
C00620=1038.929,251.970,389.972,171.152,41.873,157.986
C00621=1038.922,251.722,390.000,171.148,41.872,157.985
C00622=1038.915,251.474,390.030,171.146,41.870,157.985
C00623=1038.908,251.226,390.060,171.142,41.869,157.984
C00624=1038.902,250.978,390.089,171.140,41.868,157.984
C00625=1038.896,250.730,390.118,171.137,41.866,157.983
C00626=1038.889,250.481,390.147,171.134,41.865,157.983
C00627=1038.883,250.233,390.176,171.131,41.863,157.982
C00628=1038.875,249.986,390.205,171.129,41.862,157.982
C00629=1038.868,249.737,390.235,171.125,41.861,157.981
C00630=1038.862,249.489,390.264,171.123,41.859,157.981
C00631=1038.854,249.176,390.301,171.119,41.857,157.980
C00632=1038.846,248.864,390.337,171.115,41.856,157.980
C00633=1038.838,248.551,390.373,171.111,41.854,157.979
C00634=1038.829,248.239,390.410,171.108,41.852,157.979
C00635=1038.823,247.991,390.439,171.105,41.851,157.978
C00636=1038.816,247.743,390.468,171.103,41.849,157.978
C00637=1038.810,247.495,390.497,171.099,41.848,157.977
C00638=1038.803,247.246,390.527,171.097,41.846,157.977
C00639=1038.797,246.998,390.556,171.094,41.845,157.976
C00640=1038.791,246.750,390.585,171.092,41.844,157.976
C00641=1038.784,246.502,390.613,171.088,41.842,157.975
C00642=1038.777,246.254,390.642,171.085,41.841,157.975
C00643=1038.771,246.005,390.672,171.083,41.839,157.974
C00644=1038.764,245.757,390.701,171.079,41.838,157.974
C00645=1038.758,245.509,390.730,171.077,41.837,157.973
C00646=1038.752,245.261,390.759,171.074,41.835,157.973
C00647=1038.745,245.013,390.787,171.072,41.834,157.972
C00648=1038.738,244.764,390.817,171.068,41.832,157.972
C00649=1038.732,244.516,390.846,171.066,41.831,157.971
C00650=1038.725,244.267,390.873,171.063,41.830,157.971
C00651=1038.719,244.019,390.903,171.061,41.828,157.970
C00652=1038.711,243.771,390.931,171.057,41.827,157.970
C00653=1038.705,243.523,390.960,171.055,41.826,157.970
C00654=1038.698,243.275,390.989,171.052,41.824,157.969
C00655=1038.692,243.026,391.017,171.049,41.823,157.969
C00656=1038.686,242.778,391.046,171.046,41.822,157.968
C00657=1038.678,242.529,391.075,171.044,41.820,157.968
C00658=1038.672,242.281,391.104,171.041,41.819,157.967
C00659=1038.665,242.033,391.132,171.038,41.818,157.967
C00660=1038.659,241.785,391.161,171.035,41.816,157.966
C00661=1038.652,241.537,391.189,171.032,41.815,157.966
C00662=1038.646,241.288,391.218,171.030,41.814,157.965
C00663=1038.640,241.040,391.247,171.026,41.812,157.965
C00664=1038.632,240.791,391.275,171.024,41.811,157.964
C00665=1038.626,240.543,391.303,171.021,41.810,157.964
C00666=1038.619,240.295,391.332,171.019,41.808,157.964
C00667=1038.612,240.047,391.361,171.015,41.807,157.963
C00668=1038.606,239.799,391.388,171.013,41.806,157.963
C00669=1038.599,239.550,391.417,171.011,41.805,157.962
C00670=1038.592,239.301,391.446,171.008,41.803,157.962
C00671=1038.585,239.053,391.474,171.004,41.802,157.961
C00672=1038.579,238.805,391.502,171.002,41.801,157.961
C00673=1038.572,238.557,391.531,170.999,41.799,157.961
C00674=1038.566,238.308,391.558,170.997,41.798,157.960
C00675=1038.559,238.060,391.587,170.994,41.797,157.960
C00676=1038.553,237.812,391.615,170.991,41.795,157.959
C00677=1038.545,237.563,391.644,170.988,41.794,157.959
C00678=1038.539,237.315,391.672,170.986,41.793,157.958
C00679=1038.532,237.067,391.701,170.983,41.792,157.958
C00680=1038.525,236.818,391.729,170.980,41.790,157.957
C00681=1038.519,236.570,391.756,170.978,41.789,157.957
C00682=1038.513,236.322,391.785,170.975,41.788,157.957
C00683=1038.506,236.073,391.813,170.972,41.786,157.956
C00684=1038.499,235.825,391.841,170.970,41.785,157.956
C00685=1038.492,235.577,391.869,170.966,41.784,157.955
C00686=1038.486,235.328,391.898,170.964,41.783,157.955
C00687=1038.477,235.010,391.933,170.960,41.781,157.954
C00688=1038.469,234.692,391.970,170.958,41.779,157.954
C00689=1038.459,234.374,392.006,170.954,41.778,157.953
C00690=1038.452,234.056,392.041,170.951,41.776,157.953
C00691=1038.445,233.808,392.070,170.948,41.775,157.952
C00692=1038.438,233.560,392.098,170.946,41.774,157.952
C00693=1038.432,233.311,392.126,170.943,41.772,157.951
C00694=1038.425,233.063,392.154,170.940,41.771,157.951
C00695=1038.419,232.814,392.182,170.937,41.770,157.950
C00696=1038.412,232.566,392.210,170.934,41.768,157.950
C00697=1038.406,232.317,392.238,170.932,41.767,157.950
C00698=1038.399,232.069,392.267,170.929,41.766,157.949
C00699=1038.392,231.821,392.294,170.927,41.765,157.949
C00700=1038.386,231.573,392.322,170.925,41.763,157.948
C00701=1038.379,231.324,392.350,170.922,41.762,157.948
C00702=1038.372,231.076,392.377,170.919,41.761,157.947
C00703=1038.366,230.828,392.407,170.916,41.759,157.947
C00704=1038.359,230.579,392.434,170.914,41.758,157.947
C00705=1038.353,230.331,392.462,170.911,41.757,157.946
C00706=1038.346,230.082,392.490,170.909,41.756,157.946
C00707=1038.339,229.834,392.517,170.906,41.754,157.945
C00708=1038.333,229.585,392.545,170.904,41.753,157.945
C00709=1038.326,229.337,392.573,170.901,41.752,157.944
C00710=1038.319,229.088,392.601,170.898,41.751,157.944
C00711=1038.313,228.840,392.628,170.895,41.749,157.944
C00712=1038.306,228.592,392.656,170.893,41.748,157.943
C00713=1038.299,228.344,392.685,170.890,41.747,157.943
C00714=1038.292,228.095,392.712,170.888,41.746,157.942
C00715=1038.286,227.846,392.739,170.885,41.744,157.942
C00716=1038.279,227.598,392.767,170.883,41.743,157.942
C00717=1038.273,227.349,392.795,170.880,41.742,157.941
C00718=1038.266,227.101,392.822,170.878,41.740,157.941
C00719=1038.259,226.853,392.850,170.875,41.740,157.940
C00720=1038.252,226.604,392.877,170.872,41.738,157.940
C00721=1038.245,226.356,392.905,170.870,41.737,157.939
C00722=1038.238,226.108,392.933,170.867,41.736,157.939
C00723=1038.232,225.860,392.960,170.865,41.735,157.939
C00724=1038.226,225.611,392.988,170.862,41.734,157.938
C00725=1038.219,225.363,393.016,170.860,41.732,157.938
C00726=1038.212,225.114,393.043,170.857,41.731,157.937
C00727=1038.205,224.866,393.070,170.855,41.729,157.937
C00728=1038.198,224.617,393.098,170.852,41.728,157.937
C00729=1038.192,224.369,393.125,170.850,41.727,157.936
C00730=1038.185,224.120,393.153,170.847,41.726,157.936
C00731=1038.178,223.872,393.181,170.844,41.724,157.935
C00732=1038.172,223.624,393.208,170.841,41.724,157.935
C00733=1038.166,223.375,393.235,170.839,41.723,157.935
C00734=1038.159,223.127,393.262,170.836,41.721,157.934
C00735=1038.152,222.879,393.290,170.834,41.720,157.934
C00736=1038.145,222.630,393.318,170.831,41.718,157.933
C00737=1038.139,222.381,393.345,170.829,41.717,157.933
C00738=1038.132,222.133,393.372,170.827,41.716,157.932
C00739=1038.126,221.885,393.400,170.824,41.715,157.932
C00740=1038.119,221.637,393.427,170.822,41.713,157.932
C00741=1038.112,221.388,393.454,170.819,41.712,157.931
C00742=1038.106,221.139,393.482,170.817,41.711,157.931
C00743=1038.097,220.814,393.518,170.813,41.709,157.930
C00744=1038.088,220.488,393.553,170.810,41.708,157.930
C00745=1038.080,220.163,393.589,170.807,41.706,157.929
C00746=1038.071,219.837,393.625,170.804,41.705,157.929
C00747=1038.064,219.588,393.651,170.802,41.703,157.928
C00748=1038.057,219.340,393.679,170.799,41.702,157.928
C00749=1038.051,219.091,393.707,170.796,41.701,157.927
C00750=1038.044,218.843,393.733,170.793,41.700,157.927
C00751=1038.038,218.595,393.761,170.791,41.699,157.927
C00752=1038.030,218.346,393.787,170.789,41.698,157.926
C00753=1038.024,218.098,393.815,170.786,41.696,157.926
C00754=1038.017,217.849,393.841,170.784,41.695,157.925
C00755=1038.011,217.601,393.869,170.781,41.694,157.925
C00756=1038.004,217.352,393.896,170.779,41.693,157.925
C00757=1037.997,217.104,393.923,170.776,41.692,157.924
C00758=1037.990,216.855,393.950,170.774,41.690,157.924
C00759=1037.984,216.608,393.977,170.771,41.689,157.923
C00760=1037.977,216.358,394.004,170.769,41.688,157.923
C00761=1037.970,216.110,394.031,170.766,41.686,157.923
C00762=1037.963,215.861,394.058,170.765,41.685,157.922
C00763=1037.957,215.614,394.084,170.763,41.684,157.922
C00764=1037.950,215.365,394.111,170.760,41.683,157.921
C00765=1037.943,215.116,394.138,170.758,41.682,157.921
C00766=1037.936,214.868,394.166,170.755,41.680,157.921
C00767=1037.931,214.619,394.192,170.753,41.679,157.920
C00768=1037.923,214.371,394.219,170.750,41.678,157.920
C00769=1037.917,214.122,394.246,170.748,41.677,157.919
C00770=1037.910,213.874,394.272,170.746,41.676,157.919
C00771=1037.904,213.626,394.300,170.743,41.675,157.919
C00772=1037.897,213.377,394.327,170.741,41.673,157.918
C00773=1037.891,213.128,394.353,170.738,41.672,157.918
C00774=1037.883,212.880,394.380,170.736,41.671,157.917
C00775=1037.877,212.631,394.407,170.733,41.670,157.917
C00776=1037.870,212.383,394.433,170.731,41.669,157.917
C00777=1037.864,212.135,394.461,170.728,41.667,157.916
C00778=1037.857,211.886,394.488,170.726,41.666,157.916
C00779=1037.851,211.638,394.514,170.724,41.664,157.915
C00780=1037.843,211.390,394.541,170.722,41.663,157.915
C00781=1037.837,211.140,394.568,170.720,41.662,157.915
C00782=1037.831,210.892,394.594,170.717,41.661,157.914
C00783=1037.824,210.643,394.621,170.715,41.660,157.914
C00784=1037.817,210.395,394.649,170.712,41.659,157.914
C00785=1037.810,210.147,394.675,170.710,41.657,157.913
C00786=1037.804,209.898,394.702,170.707,41.656,157.913
C00787=1037.797,209.649,394.728,170.705,41.655,157.912
C00788=1037.790,209.401,394.754,170.702,41.654,157.912
C00789=1037.784,209.152,394.781,170.700,41.653,157.912
C00790=1037.777,208.905,394.808,170.699,41.652,157.911
C00791=1037.770,208.656,394.834,170.696,41.650,157.911
C00792=1037.764,208.407,394.861,170.694,41.649,157.910
C00793=1037.757,208.159,394.887,170.691,41.648,157.910
C00794=1037.750,207.910,394.914,170.689,41.646,157.910
C00795=1037.743,207.661,394.940,170.686,41.645,157.909
C00796=1037.737,207.413,394.967,170.684,41.644,157.909
C00797=1037.730,207.164,394.993,170.681,41.643,157.908
C00798=1037.723,206.916,395.019,170.679,41.642,157.908
C00799=1037.714,206.596,395.054,170.676,41.640,157.908
C00800=1037.706,206.276,395.088,170.674,41.639,157.907
C00801=1037.697,205.956,395.122,170.670,41.637,157.907
C00802=1037.688,205.636,395.155,170.668,41.636,157.906
C00803=1037.662,204.585,395.262,170.363,41.532,157.867
C00804=1037.656,204.337,395.287,170.360,41.531,157.867
C00805=1037.650,204.089,395.313,170.357,41.531,157.866
C00806=1037.644,203.839,395.337,170.354,41.530,157.866
C00807=1037.638,203.591,395.363,170.350,41.530,157.866
C00808=1037.632,203.342,395.388,170.347,41.529,157.865
C00809=1037.625,203.094,395.413,170.344,41.529,157.865
C00810=1037.619,202.845,395.438,170.341,41.529,157.865
C00811=1037.613,202.596,395.462,170.337,41.528,157.864
C00812=1037.607,202.348,395.488,170.335,41.528,157.864
C00813=1037.601,202.099,395.513,170.332,41.527,157.864
C00814=1037.595,201.850,395.538,170.329,41.527,157.864
C00815=1037.589,201.601,395.563,170.325,41.526,157.863
C00816=1037.583,201.352,395.588,170.322,41.526,157.863
C00817=1037.577,201.105,395.613,170.319,41.526,157.863
C00818=1037.571,200.855,395.638,170.315,41.525,157.863
C00819=1037.564,200.607,395.663,170.312,41.525,157.862
C00820=1037.558,200.358,395.688,170.309,41.524,157.862
C00821=1037.551,200.109,395.712,170.306,41.524,157.862
C00822=1037.545,199.861,395.737,170.303,41.524,157.862
C00823=1037.538,199.612,395.761,170.300,41.524,157.861
C00824=1037.533,199.364,395.786,170.297,41.523,157.861
C00825=1037.527,199.114,395.811,170.294,41.523,157.861
C00826=1037.520,198.866,395.836,170.291,41.523,157.861
C00827=1037.514,198.617,395.860,170.288,41.523,157.861
C00828=1037.507,198.368,395.885,170.284,41.522,157.860
C00829=1037.502,198.120,395.909,170.281,41.522,157.860
C00830=1037.495,197.871,395.934,170.278,41.521,157.860
C00831=1037.489,197.622,395.959,170.274,41.521,157.859
C00832=1037.482,197.374,395.983,170.271,41.521,157.859
C00833=1037.477,197.125,396.008,170.269,41.521,157.859
C00834=1037.471,196.876,396.033,170.266,41.520,157.859
C00835=1037.464,196.627,396.057,170.263,41.520,157.859
C00836=1037.458,196.378,396.082,170.259,41.520,157.858
C00837=1037.452,196.131,396.106,170.256,41.520,157.858
C00838=1037.446,195.881,396.131,170.253,41.519,157.858
C00839=1037.439,195.633,396.155,170.250,41.519,157.858
C00840=1037.433,195.384,396.180,170.247,41.519,157.857
C00841=1037.427,195.135,396.204,170.244,41.519,157.857
C00842=1037.421,194.887,396.229,170.241,41.518,157.857
C00843=1037.414,194.638,396.253,170.238,41.518,157.857
C00844=1037.409,194.389,396.277,170.235,41.518,157.857
C00845=1037.402,194.141,396.302,170.232,41.518,157.856
C00846=1037.396,193.891,396.327,170.228,41.517,157.856
C00847=1037.390,193.643,396.350,170.226,41.517,157.856
C00848=1037.384,193.394,396.376,170.223,41.517,157.856
C00849=1037.377,193.146,396.400,170.220,41.517,157.855
C00850=1037.372,192.897,396.424,170.217,41.516,157.855
C00851=1037.366,192.648,396.448,170.213,41.516,157.855
C00852=1037.359,192.399,396.473,170.210,41.516,157.855
C00853=1037.354,192.151,396.497,170.208,41.516,157.855
C00854=1037.347,191.902,396.522,170.205,41.515,157.854
C00855=1037.341,191.652,396.546,170.202,41.515,157.854
C00856=1037.335,191.405,396.571,170.198,41.515,157.854
C00857=1037.329,191.155,396.595,170.195,41.515,157.854
C00858=1037.323,190.907,396.619,170.193,41.514,157.853
C00859=1037.317,190.658,396.643,170.190,41.514,157.853
C00860=1037.310,190.409,396.667,170.186,41.514,157.853
C00861=1037.305,190.160,396.692,170.183,41.514,157.853
C00862=1037.298,189.912,396.716,170.181,41.513,157.852
C00863=1037.293,189.663,396.741,170.178,41.513,157.852
C00864=1037.286,189.379,396.768,170.175,41.513,157.852
C00865=1037.279,189.095,396.796,170.170,41.513,157.852
C00866=1037.272,188.810,396.823,170.167,41.512,157.852
C00867=1037.265,188.526,396.851,170.164,41.512,157.851
C00868=1037.258,188.278,396.875,170.161,41.512,157.851
C00869=1037.253,188.028,396.899,170.159,41.512,157.851
C00870=1037.247,187.780,396.923,170.155,41.511,157.851
C00871=1037.241,187.531,396.948,170.152,41.511,157.850
C00872=1037.235,187.283,396.971,170.149,41.511,157.850
C00873=1037.229,187.033,396.996,170.147,41.510,157.850
C00874=1037.223,186.785,397.020,170.144,41.510,157.850
C00875=1037.217,186.536,397.044,170.140,41.510,157.849
C00876=1037.211,186.287,397.068,170.137,41.510,157.849
C00877=1037.205,186.038,397.093,170.135,41.509,157.849
C00878=1037.199,185.790,397.116,170.132,41.510,157.849
C00879=1037.193,185.541,397.141,170.129,41.510,157.849
C00880=1037.187,185.292,397.165,170.127,41.509,157.849
C00881=1037.182,185.044,397.189,170.123,41.509,157.848
C00882=1037.175,184.795,397.213,170.120,41.509,157.848
C00883=1037.169,184.546,397.237,170.117,41.508,157.848
C00884=1037.163,184.297,397.261,170.115,41.508,157.848
C00885=1037.157,184.049,397.285,170.111,41.508,157.847
C00886=1037.152,183.800,397.309,170.108,41.508,157.847
C00887=1037.145,183.551,397.333,170.106,41.507,157.847
C00888=1037.140,183.302,397.357,170.103,41.508,157.847
C00889=1037.133,183.053,397.381,170.100,41.507,157.847
C00890=1037.127,182.805,397.404,170.097,41.507,157.846
C00891=1037.120,182.556,397.427,170.095,41.507,157.846
C00892=1037.114,182.307,397.451,170.091,41.507,157.846
C00893=1037.108,182.058,397.475,170.088,41.508,157.846
C00894=1037.102,181.809,397.498,170.085,41.507,157.846
C00895=1037.095,181.560,397.522,170.083,41.508,157.846
C00896=1037.089,181.312,397.545,170.080,41.507,157.845
C00897=1037.083,181.063,397.569,170.077,41.507,157.845
C00898=1037.077,180.814,397.592,170.074,41.508,157.845
C00899=1037.070,180.565,397.616,170.071,41.507,157.845
C00900=1037.064,180.317,397.639,170.068,41.508,157.845
C00901=1037.057,180.068,397.663,170.065,41.507,157.845
C00902=1037.051,179.819,397.686,170.062,41.508,157.845
C00903=1037.045,179.570,397.710,170.060,41.507,157.844
C00904=1037.039,179.321,397.733,170.057,41.507,157.844
C00905=1037.033,179.073,397.756,170.054,41.508,157.844
C00906=1037.027,178.823,397.780,170.052,41.507,157.844
C00907=1037.021,178.575,397.803,170.049,41.508,157.844
C00908=1037.013,178.326,397.826,170.045,41.507,157.843
C00909=1037.007,178.077,397.850,170.042,41.508,157.843
C00910=1037.001,177.828,397.873,170.040,41.507,157.843
C00911=1036.995,177.579,397.897,170.037,41.508,157.843
C00912=1036.989,177.330,397.920,170.034,41.508,157.843
C00913=1036.983,177.082,397.944,170.032,41.507,157.843
C00914=1036.977,176.833,397.967,170.029,41.508,157.843
C00915=1036.970,176.585,397.990,170.025,41.507,157.842
C00916=1036.964,176.335,398.013,170.023,41.508,157.842
C00917=1036.958,176.087,398.037,170.020,41.507,157.842
C00918=1036.952,175.838,398.060,170.017,41.508,157.842
C00919=1036.946,175.588,398.083,170.014,41.508,157.842
C00920=1036.940,175.340,398.107,170.012,41.508,157.842
C00921=1036.934,175.091,398.129,170.009,41.508,157.841
C00922=1036.927,174.842,398.153,170.006,41.508,157.841
C00923=1036.921,174.594,398.176,170.003,41.508,157.841
C00924=1036.915,174.345,398.199,170.000,41.508,157.841
C00925=1036.909,174.096,398.223,169.997,41.508,157.841
C00926=1036.903,173.847,398.246,169.995,41.508,157.841
C00927=1036.897,173.598,398.269,169.992,41.508,157.841
C00928=1036.889,173.313,398.295,169.989,41.508,157.840
C00929=1036.883,173.029,398.322,169.986,41.508,157.840
C00930=1036.875,172.744,398.348,169.982,41.508,157.840
C00931=1036.869,172.460,398.375,169.979,41.508,157.840
C00932=1036.862,172.211,398.398,169.976,41.508,157.840
C00933=1036.856,171.962,398.421,169.974,41.508,157.840
C00934=1036.850,171.713,398.444,169.971,41.508,157.839
C00935=1036.844,171.465,398.468,169.969,41.508,157.839
C00936=1036.839,171.216,398.491,169.966,41.508,157.839
C00937=1036.832,170.966,398.514,169.963,41.508,157.839
C00938=1036.826,170.717,398.536,169.961,41.508,157.839
C00939=1036.820,170.469,398.560,169.958,41.508,157.839
C00940=1036.814,170.220,398.583,169.955,41.508,157.838
C00941=1036.808,169.971,398.606,169.952,41.508,157.838
C00942=1036.802,169.722,398.629,169.949,41.508,157.838
C00943=1036.795,169.473,398.652,169.947,41.508,157.838
C00944=1036.790,169.224,398.675,169.944,41.508,157.838
C00945=1036.784,168.976,398.698,169.942,41.508,157.838
C00946=1036.778,168.727,398.721,169.939,41.508,157.838
C00947=1036.772,168.478,398.744,169.936,41.509,157.837
C00948=1036.765,168.229,398.767,169.933,41.508,157.837
C00949=1036.759,167.980,398.790,169.930,41.509,157.837
C00950=1036.754,167.731,398.813,169.928,41.508,157.837
C00951=1036.748,167.482,398.836,169.925,41.509,157.837
C00952=1036.742,167.234,398.859,169.923,41.508,157.837
C00953=1036.736,166.984,398.883,169.920,41.509,157.837
C00954=1036.729,166.736,398.905,169.917,41.508,157.836
C00955=1036.723,166.487,398.928,169.915,41.509,157.836
C00956=1036.718,166.238,398.951,169.911,41.508,157.836
C00957=1036.712,165.989,398.974,169.909,41.509,157.836
C00958=1036.705,165.741,398.996,169.906,41.509,157.836
C00959=1036.700,165.492,399.019,169.904,41.509,157.836
C00960=1036.694,165.243,399.042,169.901,41.509,157.836
C00961=1036.688,164.994,399.065,169.899,41.509,157.835
C00962=1036.683,164.745,399.088,169.896,41.509,157.835
C00963=1036.676,164.496,399.111,169.893,41.509,157.835
C00964=1036.670,164.247,399.134,169.891,41.509,157.835
C00965=1036.664,163.998,399.157,169.887,41.509,157.835
C00966=1036.658,163.749,399.179,169.885,41.509,157.835
C00967=1036.653,163.500,399.202,169.882,41.509,157.834
C00968=1036.646,163.251,399.225,169.880,41.509,157.834
C00969=1036.640,163.003,399.248,169.877,41.509,157.834
C00970=1036.635,162.754,399.271,169.875,41.509,157.834
C00971=1036.629,162.505,399.294,169.872,41.509,157.834
C00972=1036.622,162.256,399.316,169.870,41.509,157.834
C00973=1036.617,162.007,399.339,169.867,41.509,157.834
C00974=1036.611,161.758,399.361,169.864,41.509,157.833
C00975=1036.606,161.509,399.384,169.861,41.510,157.833
C00976=1036.599,161.260,399.406,169.859,41.509,157.833
C00977=1036.593,161.011,399.429,169.856,41.510,157.833
C00978=1036.588,160.763,399.452,169.854,41.509,157.833
C00979=1036.582,160.514,399.475,169.851,41.510,157.833
C00980=1036.576,160.265,399.498,169.849,41.509,157.833
C00981=1036.570,160.016,399.520,169.846,41.510,157.833
C00982=1036.564,159.767,399.543,169.844,41.510,157.832
C00983=1036.558,159.518,399.565,169.841,41.510,157.832
C00984=1036.551,159.269,399.588,169.839,41.510,157.832
C00985=1036.546,159.020,399.610,169.835,41.510,157.832
C00986=1036.539,158.771,399.632,169.833,41.511,157.832
C00987=1036.534,158.522,399.655,169.830,41.510,157.832
C00988=1036.528,158.273,399.677,169.828,41.511,157.832
C00989=1036.521,158.025,399.699,169.825,41.511,157.832
C00990=1036.515,157.776,399.722,169.823,41.511,157.832
C00991=1036.509,157.527,399.744,169.820,41.511,157.831
C00992=1036.502,157.241,399.770,169.817,41.512,157.831
C00993=1036.495,156.956,399.795,169.814,41.512,157.831
C00994=1036.488,156.671,399.821,169.811,41.512,157.831
C00995=1036.481,156.386,399.846,169.809,41.512,157.831
C00996=1036.475,156.137,399.868,169.806,41.512,157.831
C00997=1036.469,155.888,399.890,169.803,41.513,157.831
C00998=1036.463,155.639,399.913,169.801,41.513,157.831
C00999=1036.456,155.391,399.935,169.797,41.513,157.830
C01000=1036.451,155.141,399.957,169.795,41.513,157.830
C01001=1036.444,154.893,399.979,169.793,41.513,157.830
C01002=1036.438,154.643,400.001,169.790,41.514,157.830
C01003=1036.432,154.395,400.024,169.788,41.513,157.830
C01004=1036.426,154.145,400.046,169.785,41.514,157.830
C01005=1036.420,153.897,400.068,169.783,41.514,157.830
C01006=1036.414,153.648,400.090,169.780,41.514,157.830
C01007=1036.408,153.399,400.113,169.778,41.515,157.830
C01008=1036.402,153.149,400.134,169.775,41.515,157.829
C01009=1036.396,152.900,400.156,169.773,41.515,157.829
C01010=1036.390,152.652,400.178,169.770,41.515,157.829
C01011=1036.384,152.403,400.200,169.768,41.515,157.829
C01012=1036.378,152.154,400.222,169.765,41.516,157.829
C01013=1036.372,151.905,400.244,169.763,41.516,157.829
C01014=1036.365,151.657,400.266,169.760,41.516,157.829
C01015=1036.359,151.407,400.288,169.758,41.517,157.829
C01016=1036.353,151.158,400.310,169.754,41.516,157.829
C01017=1036.346,150.910,400.332,169.752,41.517,157.829
C01018=1036.341,150.660,400.354,169.749,41.517,157.828
C01019=1036.335,150.411,400.376,169.747,41.517,157.828
C01020=1036.329,150.163,400.398,169.744,41.518,157.828
C01021=1036.323,149.914,400.420,169.742,41.518,157.828
C01022=1036.317,149.664,400.441,169.739,41.518,157.828
C01023=1036.310,149.416,400.464,169.737,41.518,157.828
C01024=1036.305,149.166,400.486,169.735,41.518,157.828
C01025=1036.299,148.917,400.507,169.732,41.519,157.828
C01026=1036.292,148.669,400.530,169.730,41.519,157.828
C01027=1036.286,148.419,400.551,169.727,41.519,157.828
C01028=1036.280,148.171,400.573,169.725,41.520,157.828
C01029=1036.274,147.922,400.594,169.722,41.520,157.827
C01030=1036.268,147.673,400.617,169.720,41.520,157.827
C01031=1036.262,147.424,400.638,169.716,41.520,157.827
C01032=1036.255,147.175,400.660,169.714,41.520,157.827
C01033=1036.250,146.925,400.682,169.711,41.521,157.827
C01034=1036.244,146.677,400.703,169.709,41.521,157.827
C01035=1036.237,146.428,400.725,169.707,41.521,157.827
C01036=1036.231,146.179,400.747,169.704,41.522,157.827
C01037=1036.225,145.930,400.768,169.702,41.522,157.827
C01038=1036.219,145.681,400.790,169.699,41.522,157.827
C01039=1036.213,145.432,400.812,169.697,41.523,157.827
C01040=1036.206,145.182,400.833,169.694,41.523,157.826
C01041=1036.201,144.934,400.855,169.692,41.523,157.826
C01042=1036.195,144.685,400.876,169.689,41.524,157.826
C01043=1036.188,144.436,400.899,169.687,41.524,157.826
C01044=1036.182,144.187,400.920,169.685,41.524,157.826
C01045=1036.176,143.938,400.942,169.682,41.525,157.826
C01046=1036.170,143.689,400.963,169.680,41.525,157.826
C01047=1036.163,143.440,400.984,169.677,41.525,157.826
C01048=1036.157,143.191,401.006,169.675,41.525,157.826
C01049=1036.151,142.942,401.027,169.672,41.526,157.826
C01050=1036.146,142.693,401.049,169.670,41.526,157.826
C01051=1036.139,142.444,401.070,169.668,41.526,157.826
C01052=1036.133,142.195,401.092,169.665,41.527,157.825
C01053=1036.127,141.946,401.114,169.663,41.526,157.825
C01054=1036.121,141.697,401.135,169.660,41.527,157.825
C01055=1036.115,141.448,401.157,169.658,41.527,157.825
C01056=1036.107,141.163,401.181,169.655,41.527,157.825
C01057=1036.101,140.877,401.206,169.652,41.528,157.825
C01058=1036.095,140.592,401.231,169.650,41.528,157.825
C01059=1036.087,140.306,401.255,169.646,41.529,157.825
C01060=1036.081,140.058,401.277,169.643,41.529,157.825
C01061=1036.075,139.808,401.297,169.641,41.529,157.825
C01062=1036.069,139.559,401.319,169.639,41.529,157.825
C01063=1036.064,139.310,401.340,169.636,41.530,157.824
C01064=1036.057,139.061,401.361,169.634,41.530,157.824
C01065=1036.050,138.812,401.383,169.631,41.530,157.824
C01066=1036.044,138.563,401.405,169.629,41.531,157.824
C01067=1036.039,138.314,401.426,169.627,41.531,157.824
C01068=1036.032,138.066,401.447,169.624,41.531,157.824
C01069=1036.026,137.816,401.468,169.622,41.532,157.824
C01070=1036.020,137.567,401.489,169.619,41.532,157.824
C01071=1036.014,137.318,401.511,169.617,41.532,157.824
C01072=1036.007,137.069,401.532,169.615,41.533,157.824
C01073=1036.002,136.821,401.553,169.612,41.534,157.824
C01074=1035.996,136.571,401.574,169.610,41.534,157.824
C01075=1035.989,136.322,401.595,169.607,41.534,157.824
C01076=1035.983,136.073,401.617,169.605,41.535,157.824
C01077=1035.977,135.824,401.638,169.603,41.535,157.824
C01078=1035.971,135.575,401.658,169.600,41.535,157.823
C01079=1035.965,135.325,401.680,169.598,41.536,157.823
C01080=1035.959,135.077,401.701,169.595,41.536,157.823
C01081=1035.952,134.828,401.722,169.593,41.536,157.823
C01082=1035.946,134.578,401.743,169.591,41.536,157.823
C01083=1035.941,134.330,401.764,169.588,41.537,157.823
C01084=1035.934,134.081,401.785,169.586,41.537,157.823
C01085=1035.928,133.832,401.806,169.584,41.537,157.823
C01086=1035.922,133.582,401.828,169.581,41.538,157.823
C01087=1035.915,133.334,401.849,169.579,41.539,157.823
C01088=1035.910,133.084,401.869,169.576,41.539,157.823
C01089=1035.903,132.836,401.890,169.574,41.539,157.823
C01090=1035.897,132.586,401.912,169.572,41.540,157.823
C01091=1035.892,132.337,401.932,169.569,41.540,157.823
C01092=1035.885,132.088,401.954,169.567,41.540,157.822
C01093=1035.879,131.840,401.975,169.565,41.541,157.822
C01094=1035.874,131.590,401.996,169.562,41.541,157.822
C01095=1035.867,131.341,402.017,169.560,41.541,157.822
C01096=1035.861,131.092,402.037,169.558,41.541,157.822
C01097=1035.854,130.843,402.058,169.555,41.542,157.822
C01098=1035.849,130.594,402.079,169.553,41.542,157.822
C01099=1035.842,130.345,402.100,169.550,41.543,157.822
C01100=1035.836,130.096,402.120,169.548,41.543,157.822
C01101=1035.830,129.847,402.142,169.546,41.544,157.822
C01102=1035.824,129.598,402.162,169.543,41.544,157.822
C01103=1035.817,129.349,402.183,169.541,41.545,157.822
C01104=1035.811,129.100,402.203,169.538,41.545,157.822
C01105=1035.805,128.851,402.224,169.536,41.546,157.822
C01106=1035.799,128.602,402.244,169.534,41.546,157.822
C01107=1035.792,128.353,402.266,169.531,41.547,157.822
C01108=1035.786,128.103,402.286,169.529,41.547,157.822
C01109=1035.780,127.854,402.306,169.527,41.547,157.822
C01110=1035.774,127.605,402.328,169.524,41.548,157.821
C01111=1035.768,127.356,402.348,169.522,41.548,157.821
C01112=1035.761,127.107,402.369,169.519,41.549,157.821
C01113=1035.755,126.859,402.389,169.517,41.549,157.821
C01114=1035.749,126.609,402.410,169.515,41.550,157.821
C01115=1035.742,126.360,402.431,169.512,41.550,157.821
C01116=1035.736,126.111,402.451,169.510,41.550,157.821
C01117=1035.730,125.861,402.472,169.508,41.551,157.821
C01118=1035.724,125.613,402.492,169.505,41.552,157.821
C01119=1035.717,125.364,402.513,169.503,41.552,157.821
C01120=1035.710,125.078,402.536,169.500,41.552,157.821
C01121=1035.703,124.793,402.560,169.498,41.553,157.821
C01122=1035.696,124.507,402.584,169.495,41.554,157.821
C01123=1035.689,124.222,402.607,169.492,41.554,157.821
C01124=1035.683,123.972,402.628,169.490,41.554,157.821
C01125=1035.677,123.723,402.648,169.487,41.555,157.821
C01126=1035.671,123.474,402.669,169.485,41.556,157.821
C01127=1035.664,123.226,402.689,169.483,41.556,157.821
C01128=1035.658,122.976,402.710,169.480,41.556,157.821
C01129=1035.653,122.727,402.730,169.478,41.557,157.821
C01130=1035.646,122.477,402.751,169.476,41.557,157.820
C01131=1035.640,122.229,402.771,169.473,41.558,157.820
C01132=1035.634,121.979,402.792,169.471,41.558,157.820
C01133=1035.628,121.731,402.812,169.469,41.558,157.820
C01134=1035.621,121.481,402.832,169.466,41.559,157.820
C01135=1035.615,121.233,402.853,169.464,41.559,157.820
C01136=1035.609,120.983,402.874,169.462,41.560,157.820
C01137=1035.603,120.734,402.894,169.460,41.560,157.820
C01138=1035.597,120.485,402.914,169.457,41.561,157.820
C01139=1035.591,120.236,402.934,169.455,41.561,157.820
C01140=1035.585,119.987,402.955,169.453,41.561,157.820
C01141=1035.578,119.738,402.976,169.450,41.562,157.820
C01142=1035.572,119.489,402.996,169.448,41.562,157.820
C01143=1035.566,119.239,403.017,169.446,41.563,157.820
C01144=1035.561,118.990,403.037,169.443,41.563,157.820
C01145=1035.555,118.742,403.057,169.441,41.563,157.820
C01146=1035.548,118.492,403.077,169.439,41.564,157.820
C01147=1035.543,118.243,403.097,169.436,41.565,157.820
C01148=1035.536,117.994,403.119,169.434,41.565,157.820
C01149=1035.530,117.745,403.138,169.432,41.565,157.820
C01150=1035.524,117.497,403.158,169.430,41.566,157.819
C01151=1035.518,117.247,403.179,169.427,41.566,157.819
C01152=1035.512,116.998,403.199,169.425,41.566,157.819
C01153=1035.506,116.749,403.219,169.423,41.567,157.819
C01154=1035.499,116.500,403.240,169.420,41.568,157.819
C01155=1035.494,116.250,403.260,169.418,41.568,157.819
C01156=1035.488,116.002,403.280,169.416,41.568,157.819
C01157=1035.481,115.752,403.300,169.414,41.568,157.819
C01158=1035.475,115.503,403.320,169.411,41.569,157.819
C01159=1035.470,115.254,403.341,169.409,41.570,157.819
C01160=1035.464,115.005,403.361,169.407,41.570,157.819
C01161=1035.458,114.756,403.381,169.405,41.570,157.819
C01162=1035.452,114.507,403.401,169.402,41.571,157.819
C01163=1035.446,114.257,403.422,169.400,41.571,157.819
C01164=1035.440,114.008,403.442,169.398,41.571,157.819
C01165=1035.434,113.760,403.462,169.396,41.571,157.819
C01166=1035.427,113.510,403.482,169.393,41.572,157.819
C01167=1035.422,113.261,403.503,169.391,41.573,157.819
C01168=1035.415,113.012,403.522,169.389,41.573,157.819
C01169=1035.409,112.763,403.543,169.386,41.573,157.818
C01170=1035.403,112.514,403.563,169.384,41.574,157.818
C01171=1035.396,112.265,403.583,169.382,41.574,157.818
C01172=1035.390,112.016,403.603,169.379,41.575,157.818
C01173=1035.384,111.766,403.622,169.377,41.575,157.818
C01174=1035.378,111.518,403.642,169.375,41.576,157.818
C01175=1035.372,111.268,403.662,169.373,41.576,157.818
C01176=1035.366,111.019,403.682,169.370,41.577,157.818
C01177=1035.360,110.770,403.702,169.368,41.578,157.818
C01178=1035.353,110.520,403.722,169.366,41.578,157.818
C01179=1035.347,110.271,403.742,169.363,41.578,157.818
C01180=1035.342,110.023,403.762,169.361,41.579,157.818
C01181=1035.335,109.773,403.782,169.359,41.579,157.818
C01182=1035.329,109.524,403.802,169.357,41.580,157.818
C01183=1035.322,109.275,403.821,169.354,41.581,157.818
C01184=1035.316,108.989,403.844,169.352,41.581,157.818
C01185=1035.308,108.703,403.866,169.349,41.581,157.818
C01186=1035.301,108.418,403.890,169.347,41.583,157.818
C01187=1035.294,108.132,403.912,169.344,41.583,157.818
C01188=1035.288,107.882,403.932,169.342,41.584,157.818
C01189=1035.282,107.633,403.952,169.340,41.584,157.818
C01190=1035.275,107.385,403.971,169.338,41.584,157.818
C01191=1035.269,107.135,403.990,169.336,41.585,157.818
C01192=1035.263,106.886,404.011,169.333,41.586,157.818
C01193=1035.257,106.637,404.031,169.331,41.586,157.818
C01194=1035.251,106.388,404.050,169.329,41.587,157.818
C01195=1035.244,106.139,404.069,169.326,41.587,157.818
C01196=1035.238,105.890,404.089,169.324,41.588,157.818
C01197=1035.232,105.640,404.109,169.322,41.588,157.818
C01198=1035.226,105.391,404.129,169.320,41.589,157.818
C01199=1035.220,105.142,404.148,169.317,41.589,157.817
C01200=1035.213,104.893,404.168,169.315,41.590,157.818
C01201=1035.207,104.644,404.188,169.313,41.590,157.817
C01202=1035.201,104.395,404.207,169.310,41.591,157.817
C01203=1035.195,104.146,404.227,169.308,41.592,157.817
C01204=1035.188,103.896,404.246,169.306,41.592,157.817
C01205=1035.182,103.647,404.266,169.304,41.592,157.817
C01206=1035.176,103.398,404.286,169.301,41.593,157.817
C01207=1035.171,103.149,404.305,169.299,41.593,157.817
C01208=1035.165,102.900,404.325,169.297,41.594,157.817
C01209=1035.157,102.650,404.344,169.295,41.594,157.817
C01210=1035.151,102.401,404.364,169.292,41.595,157.817
C01211=1035.146,102.152,404.383,169.290,41.595,157.817
C01212=1035.140,101.903,404.403,169.288,41.596,157.817
C01213=1035.133,101.654,404.422,169.286,41.596,157.817
C01214=1035.127,101.405,404.442,169.283,41.597,157.817
C01215=1035.121,101.155,404.461,169.281,41.597,157.817
C01216=1035.115,100.906,404.481,169.279,41.598,157.817
C01217=1035.109,100.657,404.500,169.277,41.598,157.817
C01218=1035.103,100.408,404.520,169.274,41.599,157.817
C01219=1035.097,100.159,404.539,169.272,41.599,157.817
C01220=1035.091,99.910,404.559,169.270,41.600,157.817
C01221=1035.085,99.661,404.578,169.268,41.600,157.817
C01222=1035.078,99.411,404.597,169.266,41.601,157.817
C01223=1035.072,99.162,404.617,169.264,41.601,157.817
C01224=1035.066,98.913,404.636,169.262,41.602,157.817
C01225=1035.059,98.664,404.655,169.259,41.603,157.817
C01226=1035.053,98.415,404.675,169.257,41.603,157.817
C01227=1035.046,98.165,404.694,169.255,41.604,157.817
C01228=1035.041,97.916,404.713,169.253,41.604,157.817
C01229=1035.034,97.667,404.732,169.250,41.605,157.817
C01230=1035.028,97.418,404.751,169.248,41.606,157.817
C01231=1035.022,97.169,404.770,169.246,41.606,157.817
C01232=1035.016,96.920,404.790,169.243,41.607,157.817
C01233=1035.009,96.671,404.809,169.241,41.607,157.816
C01234=1035.004,96.421,404.828,169.239,41.608,157.817
C01235=1034.996,96.172,404.848,169.237,41.608,157.816
C01236=1034.991,95.923,404.867,169.234,41.609,157.817
C01237=1034.984,95.674,404.886,169.232,41.610,157.816
C01238=1034.979,95.424,404.905,169.230,41.610,157.816
C01239=1034.972,95.176,404.924,169.228,41.611,157.816
C01240=1034.965,94.926,404.943,169.225,41.611,157.816
C01241=1034.960,94.677,404.962,169.223,41.612,157.816
C01242=1034.953,94.428,404.981,169.221,41.612,157.816
C01243=1034.947,94.179,405.001,169.219,41.613,157.816
C01244=1034.941,93.930,405.019,169.216,41.614,157.816
C01245=1034.935,93.680,405.039,169.214,41.614,157.816
C01246=1034.928,93.431,405.058,169.212,41.614,157.816
C01247=1034.923,93.181,405.077,169.211,41.615,157.816
C01248=1034.916,92.896,405.099,169.208,41.616,157.816
C01249=1034.909,92.610,405.120,169.205,41.617,157.816
C01250=1034.901,92.324,405.143,169.203,41.617,157.816
C01251=1034.895,92.039,405.164,169.200,41.618,157.816
C01252=1034.888,91.790,405.183,169.198,41.618,157.816
C01253=1034.882,91.541,405.203,169.196,41.618,157.816
C01254=1034.876,91.292,405.221,169.194,41.619,157.816
C01255=1034.870,91.042,405.241,169.191,41.620,157.816
C01256=1034.864,90.793,405.259,169.189,41.620,157.816
C01257=1034.858,90.544,405.278,169.187,41.621,157.816
C01258=1034.852,90.294,405.297,169.185,41.621,157.816
C01259=1034.846,90.045,405.316,169.182,41.622,157.816
C01260=1034.839,89.797,405.336,169.180,41.623,157.816
C01261=1034.832,89.547,405.355,169.178,41.623,157.816
C01262=1034.826,89.298,405.373,169.176,41.624,157.816
C01263=1034.820,89.048,405.393,169.173,41.624,157.816
C01264=1034.814,88.799,405.411,169.171,41.625,157.816
C01265=1034.807,88.550,405.430,169.169,41.625,157.816
C01266=1034.801,88.301,405.449,169.166,41.626,157.816
C01267=1034.795,88.051,405.466,169.164,41.627,157.816
C01268=1034.788,87.802,405.485,169.162,41.628,157.816
C01269=1034.782,87.553,405.504,169.160,41.628,157.816
C01270=1034.776,87.303,405.523,169.158,41.629,157.816
C01271=1034.770,87.054,405.542,169.156,41.629,157.816
C01272=1034.763,86.805,405.560,169.154,41.630,157.816
C01273=1034.757,86.556,405.579,169.152,41.630,157.816
C01274=1034.751,86.307,405.598,169.149,41.631,157.816
C01275=1034.745,86.057,405.617,169.147,41.632,157.816
C01276=1034.738,85.808,405.635,169.145,41.633,157.816
C01277=1034.732,85.559,405.654,169.142,41.633,157.816
C01278=1034.725,85.310,405.673,169.140,41.634,157.816
C01279=1034.719,85.061,405.691,169.138,41.634,157.816
C01280=1034.714,84.811,405.710,169.136,41.635,157.816
C01281=1034.707,84.562,405.729,169.133,41.635,157.816
C01282=1034.701,84.313,405.747,169.131,41.636,157.816
C01283=1034.694,84.064,405.766,169.129,41.637,157.816
C01284=1034.688,83.815,405.784,169.127,41.638,157.816
C01285=1034.682,83.566,405.803,169.124,41.638,157.816
C01286=1034.676,83.317,405.822,169.122,41.639,157.816
C01287=1034.670,83.067,405.840,169.120,41.639,157.816
C01288=1034.664,82.818,405.859,169.118,41.639,157.815
C01289=1034.657,82.569,405.877,169.116,41.640,157.815
C01290=1034.651,82.319,405.896,169.114,41.641,157.815
C01291=1034.645,82.070,405.915,169.112,41.642,157.815
C01292=1034.639,81.821,405.934,169.110,41.642,157.815
C01293=1034.633,81.571,405.952,169.107,41.643,157.815
C01294=1034.626,81.322,405.970,169.105,41.643,157.815
C01295=1034.620,81.073,405.989,169.103,41.644,157.815
C01296=1034.614,80.825,406.007,169.101,41.644,157.815
C01297=1034.608,80.575,406.025,169.099,41.645,157.815
C01298=1034.601,80.326,406.044,169.096,41.646,157.815
C01299=1034.596,80.076,406.063,169.094,41.646,157.815
C01300=1034.589,79.827,406.082,169.092,41.647,157.815
C01301=1034.583,79.577,406.100,169.090,41.647,157.815
C01302=1034.577,79.328,406.118,169.087,41.648,157.815
C01303=1034.570,79.079,406.137,169.085,41.649,157.815
C01304=1034.565,78.831,406.155,169.083,41.649,157.815
C01305=1034.558,78.581,406.173,169.081,41.650,157.815
C01306=1034.553,78.332,406.193,169.078,41.650,157.815
C01307=1034.546,78.082,406.211,169.076,41.651,157.815
C01308=1034.540,77.833,406.229,169.074,41.651,157.815
C01309=1034.534,77.584,406.248,169.073,41.652,157.815
C01310=1034.528,77.334,406.266,169.069,41.653,157.815
C01311=1034.521,77.085,406.284,169.068,41.654,157.815
C01312=1034.514,76.799,406.305,169.066,41.654,157.815
C01313=1034.507,76.514,406.326,169.063,41.655,157.815
C01314=1034.500,76.228,406.347,169.060,41.655,157.815
C01315=1034.493,75.942,406.367,169.058,41.656,157.815
C01316=1034.486,75.693,406.386,169.056,41.656,157.815
C01317=1034.480,75.444,406.405,169.053,41.658,157.815
C01318=1034.474,75.194,406.422,169.051,41.658,157.815
C01319=1034.467,74.945,406.441,169.049,41.659,157.815
C01320=1034.462,74.696,406.459,169.046,41.660,157.815
C01321=1034.455,74.447,406.477,169.044,41.660,157.815
C01322=1034.448,74.197,406.495,169.042,41.661,157.815
C01323=1034.442,73.948,406.513,169.040,41.661,157.815
C01324=1034.436,73.698,406.531,169.037,41.662,157.815
C01325=1034.429,73.449,406.550,169.035,41.663,157.815
C01326=1034.424,73.200,406.567,169.034,41.663,157.815
C01327=1034.417,72.951,406.586,169.032,41.664,157.815
C01328=1034.411,72.702,406.603,169.029,41.665,157.815
C01329=1034.404,72.452,406.622,169.027,41.665,157.815
C01330=1034.399,72.203,406.640,169.025,41.666,157.815
C01331=1034.393,71.954,406.658,169.023,41.666,157.815
C01332=1034.386,71.705,406.676,169.020,41.667,157.815
C01333=1034.380,71.455,406.694,169.018,41.668,157.815
C01334=1034.374,71.206,406.713,169.016,41.668,157.815
C01335=1034.367,70.957,406.730,169.014,41.669,157.815
C01336=1034.361,70.708,406.748,169.011,41.670,157.815
C01337=1034.355,70.458,406.766,169.009,41.670,157.815
C01338=1034.349,70.208,406.784,169.007,41.671,157.815
C01339=1034.343,69.960,406.803,169.005,41.671,157.815
C01340=1034.337,69.710,406.821,169.002,41.672,157.815
C01341=1034.330,69.461,406.838,169.000,41.673,157.815
C01342=1034.323,69.212,406.857,168.998,41.674,157.815
C01343=1034.318,68.963,406.874,168.996,41.674,157.815
C01344=1034.312,68.713,406.892,168.994,41.675,157.815
C01345=1034.305,68.464,406.910,168.992,41.675,157.815
C01346=1034.299,68.214,406.928,168.990,41.676,157.815
C01347=1034.293,67.965,406.946,168.988,41.677,157.815
C01348=1034.286,67.716,406.964,168.985,41.677,157.815
C01349=1034.280,67.467,406.982,168.983,41.678,157.815
C01350=1034.274,67.217,406.999,168.981,41.679,157.815
C01351=1034.267,66.968,407.016,168.979,41.679,157.815
C01352=1034.261,66.719,407.035,168.976,41.680,157.815
C01353=1034.255,66.469,407.053,168.974,41.681,157.815
C01354=1034.249,66.221,407.070,168.972,41.681,157.815
C01355=1034.242,65.971,407.088,168.969,41.682,157.815
C01356=1034.236,65.722,407.107,168.967,41.683,157.815
C01357=1034.229,65.472,407.124,168.965,41.683,157.815
C01358=1034.224,65.223,407.142,168.964,41.684,157.815
C01359=1034.218,64.974,407.159,168.961,41.685,157.815
C01360=1034.211,64.724,407.177,168.959,41.686,157.815
C01361=1034.205,64.476,407.195,168.957,41.686,157.815
C01362=1034.198,64.226,407.212,168.955,41.687,157.815
C01363=1034.192,63.977,407.230,168.952,41.687,157.815
C01364=1034.186,63.727,407.248,168.950,41.688,157.815
C01365=1034.179,63.478,407.265,168.948,41.689,157.815
C01366=1034.173,63.228,407.283,168.946,41.689,157.815
C01367=1034.166,62.979,407.301,168.943,41.690,157.815
C01368=1034.160,62.730,407.317,168.941,41.691,157.815
C01369=1034.154,62.480,407.335,168.939,41.692,157.815
C01370=1034.147,62.231,407.353,168.936,41.693,157.815
C01371=1034.141,61.982,407.370,168.935,41.694,157.815
C01372=1034.135,61.733,407.388,168.933,41.694,157.815
C01373=1034.128,61.484,407.406,168.930,41.695,157.815
C01374=1034.121,61.235,407.423,168.928,41.696,157.815
C01375=1034.115,60.985,407.441,168.926,41.697,157.815
C01376=1034.108,60.699,407.461,168.923,41.697,157.815
C01377=1034.100,60.413,407.480,168.920,41.698,157.815
C01378=1034.093,60.127,407.500,168.918,41.699,157.815
C01379=1034.086,59.841,407.520,168.915,41.700,157.815
C01380=1034.079,59.592,407.538,168.913,41.700,157.815
C01381=1034.073,59.342,407.555,168.911,41.701,157.815
C01382=1034.067,59.093,407.572,168.909,41.702,157.815
C01383=1034.060,58.844,407.590,168.907,41.703,157.815
C01384=1034.054,58.594,407.608,168.905,41.704,157.815
C01385=1034.048,58.345,407.625,168.902,41.705,157.815
C01386=1034.041,58.096,407.642,168.900,41.705,157.815
C01387=1034.036,57.846,407.659,168.898,41.706,157.815
C01388=1034.029,57.597,407.676,168.895,41.707,157.815
C01389=1034.022,57.347,407.694,168.893,41.707,157.815
C01390=1034.016,57.098,407.711,168.891,41.708,157.815
C01391=1034.010,56.849,407.728,168.889,41.709,157.815
C01392=1034.003,56.600,407.745,168.886,41.709,157.815
C01393=1033.996,56.351,407.763,168.884,41.710,157.815
C01394=1033.990,56.101,407.781,168.883,41.711,157.815
C01395=1033.984,55.852,407.798,168.880,41.712,157.815
C01396=1033.977,55.602,407.814,168.878,41.713,157.815
C01397=1033.972,55.353,407.832,168.876,41.713,157.815
C01398=1033.965,55.104,407.849,168.873,41.714,157.815
C01399=1033.958,54.854,407.867,168.871,41.715,157.815
C01400=1033.953,54.605,407.884,168.869,41.715,157.815
C01401=1033.946,54.356,407.901,168.867,41.716,157.815
C01402=1033.940,54.106,407.918,168.864,41.717,157.815
C01403=1033.934,53.857,407.936,168.862,41.717,157.815
C01404=1033.928,53.608,407.953,168.860,41.718,157.815
C01405=1033.921,53.359,407.970,168.857,41.719,157.815
C01406=1033.915,53.110,407.987,168.855,41.720,157.815
C01407=1033.909,52.859,408.004,168.854,41.721,157.815
C01408=1033.902,52.611,408.021,168.852,41.721,157.815
C01409=1033.895,52.361,408.038,168.849,41.722,157.815
C01410=1033.890,52.112,408.056,168.847,41.722,157.815
C01411=1033.883,51.862,408.073,168.845,41.723,157.815
C01412=1033.877,51.614,408.090,168.842,41.724,157.815
C01413=1033.871,51.364,408.108,168.840,41.724,157.815
C01414=1033.865,51.115,408.124,168.838,41.725,157.815
C01415=1033.858,50.865,408.141,168.836,41.726,157.815
C01416=1033.853,50.616,408.159,168.833,41.727,157.815
C01417=1033.846,50.367,408.176,168.831,41.727,157.815
C01418=1033.840,50.118,408.193,168.829,41.728,157.815
C01419=1033.833,49.868,408.210,168.826,41.729,157.815
C01420=1033.828,49.619,408.227,168.824,41.729,157.815
C01421=1033.821,49.369,408.245,168.823,41.730,157.815
C01422=1033.815,49.120,408.261,168.820,41.730,157.815
C01423=1033.809,48.870,408.279,168.818,41.731,157.815
C01424=1033.802,48.621,408.296,168.816,41.732,157.815
C01425=1033.796,48.372,408.312,168.814,41.733,157.815
C01426=1033.790,48.123,408.329,168.812,41.734,157.815
C01427=1033.784,47.874,408.347,168.809,41.734,157.815
C01428=1033.777,47.624,408.363,168.807,41.735,157.815
C01429=1033.771,47.375,408.380,168.805,41.735,157.815
C01430=1033.765,47.125,408.397,168.802,41.736,157.815
C01431=1033.759,46.876,408.415,168.800,41.737,157.815
C01432=1033.753,46.627,408.432,168.798,41.737,157.815
C01433=1033.746,46.377,408.448,168.796,41.738,157.815
C01434=1033.741,46.128,408.466,168.793,41.739,157.815
C01435=1033.734,45.878,408.482,168.791,41.739,157.815
C01436=1033.728,45.629,408.499,168.789,41.740,157.815
C01437=1033.722,45.380,408.516,168.787,41.740,157.815
C01438=1033.716,45.130,408.534,168.785,41.741,157.815
C01439=1033.710,44.881,408.551,168.783,41.742,157.815
C01440=1033.703,44.595,408.570,168.780,41.743,157.815
C01441=1033.695,44.309,408.589,168.778,41.744,157.815
C01442=1033.688,44.022,408.609,168.775,41.744,157.815
C01443=1033.681,43.735,408.628,168.773,41.745,157.815
C01444=1033.675,43.487,408.645,168.770,41.745,157.815
C01445=1033.669,43.237,408.661,168.768,41.746,157.815
C01446=1033.663,42.988,408.679,168.766,41.746,157.815
C01447=1033.657,42.738,408.695,168.763,41.748,157.815
C01448=1033.650,42.489,408.713,168.761,41.748,157.815
C01449=1033.644,42.239,408.729,168.759,41.749,157.815
C01450=1033.638,41.990,408.745,168.756,41.750,157.815
C01451=1033.631,41.741,408.763,168.755,41.751,157.815
C01452=1033.626,41.491,408.779,168.752,41.751,157.815
C01453=1033.619,41.243,408.796,168.750,41.752,157.815
C01454=1033.613,40.992,408.812,168.748,41.753,157.815
C01455=1033.607,40.743,408.829,168.746,41.753,157.815
C01456=1033.600,40.494,408.846,168.744,41.754,157.815
C01457=1033.594,40.244,408.862,168.741,41.755,157.815
C01458=1033.588,39.995,408.879,168.739,41.756,157.815
C01459=1033.581,39.746,408.896,168.737,41.756,157.815
C01460=1033.575,39.496,408.912,168.734,41.757,157.815
C01461=1033.569,39.247,408.928,168.732,41.758,157.815
C01462=1033.563,38.998,408.945,168.730,41.759,157.815
C01463=1033.556,38.748,408.962,168.727,41.759,157.815
C01464=1033.550,38.499,408.978,168.725,41.760,157.815
C01465=1033.543,38.250,408.995,168.723,41.760,157.815
C01466=1033.537,38.000,409.011,168.721,41.761,157.815
C01467=1033.531,37.751,409.028,168.719,41.762,157.815
C01468=1033.525,37.502,409.044,168.717,41.763,157.815
C01469=1033.518,37.252,409.061,168.714,41.764,157.815
C01470=1033.512,37.003,409.077,168.712,41.765,157.815
C01471=1033.506,36.753,409.094,168.710,41.765,157.815
C01472=1033.500,36.503,409.110,168.707,41.766,157.815
C01473=1033.494,36.254,409.126,168.705,41.767,157.815
C01474=1033.487,36.006,409.143,168.703,41.768,157.815
C01475=1033.480,35.756,409.159,168.700,41.768,157.815
C01476=1033.474,35.506,409.176,168.698,41.769,157.815
C01477=1033.468,35.257,409.192,168.697,41.770,157.815
C01478=1033.462,35.008,409.208,168.694,41.770,157.815
C01479=1033.455,34.758,409.224,168.692,41.771,157.815
C01480=1033.449,34.509,409.241,168.690,41.772,157.815
C01481=1033.443,34.260,409.258,168.687,41.773,157.815
C01482=1033.436,34.011,409.273,168.685,41.774,157.815
C01483=1033.430,33.761,409.290,168.682,41.775,157.815
C01484=1033.424,33.511,409.306,168.680,41.776,157.815
C01485=1033.418,33.262,409.322,168.678,41.776,157.815
C01486=1033.410,33.012,409.338,168.675,41.777,157.815
C01487=1033.404,32.763,409.355,168.674,41.778,157.815
C01488=1033.399,32.514,409.371,168.672,41.779,157.815
C01489=1033.393,32.264,409.387,168.669,41.779,157.815
C01490=1033.386,32.015,409.403,168.667,41.780,157.815
C01491=1033.379,31.766,409.420,168.665,41.781,157.815
C01492=1033.373,31.516,409.436,168.662,41.782,157.815
C01493=1033.366,31.267,409.452,168.660,41.782,157.815
C01494=1033.360,31.018,409.468,168.658,41.783,157.815
C01495=1033.354,30.768,409.485,168.655,41.784,157.815
C01496=1033.348,30.519,409.501,168.653,41.785,157.815
C01497=1033.341,30.270,409.517,168.651,41.786,157.815
C01498=1033.335,30.020,409.533,168.648,41.786,157.815
C01499=1033.329,29.771,409.549,168.647,41.787,157.815
C01500=1033.323,29.522,409.566,168.644,41.788,157.815
C01501=1033.316,29.272,409.582,168.642,41.788,157.815
C01502=1033.310,29.022,409.598,168.640,41.789,157.815
C01503=1033.304,28.773,409.614,168.637,41.790,157.815
C01504=1033.297,28.486,409.632,168.635,41.791,157.815
C01505=1033.290,28.200,409.651,168.632,41.792,157.815
C01506=1033.282,27.914,409.669,168.629,41.793,157.815
C01507=1033.275,27.627,409.687,168.627,41.794,157.815
C01508=1033.269,27.378,409.703,168.624,41.795,157.815
C01509=1033.263,27.128,409.719,168.622,41.795,157.815
C01510=1033.257,26.879,409.735,168.620,41.796,157.815
C01511=1033.250,26.630,409.751,168.618,41.797,157.815
C01512=1033.244,26.381,409.767,168.616,41.798,157.815
C01513=1033.237,26.131,409.783,168.613,41.798,157.815
C01514=1033.231,25.881,409.799,168.611,41.799,157.815
C01515=1033.224,25.632,409.815,168.608,41.800,157.815
C01516=1033.218,25.383,409.831,168.606,41.801,157.815
C01517=1033.212,25.134,409.847,168.604,41.802,157.815
C01518=1033.206,24.884,409.863,168.601,41.803,157.815
C01519=1033.199,24.635,409.878,168.599,41.804,157.815
C01520=1033.193,24.385,409.894,168.598,41.804,157.815
C01521=1033.186,24.136,409.910,168.595,41.806,157.815
C01522=1033.180,23.886,409.926,168.593,41.806,157.815
C01523=1033.174,23.637,409.942,168.590,41.807,157.815
C01524=1033.168,23.387,409.957,168.588,41.808,157.815
C01525=1033.161,23.138,409.973,168.586,41.809,157.815
C01526=1033.155,22.889,409.989,168.583,41.809,157.815
C01527=1033.149,22.639,410.004,168.581,41.810,157.815
C01528=1033.143,22.390,410.021,168.578,41.811,157.815
C01529=1033.136,22.140,410.037,168.576,41.811,157.815
C01530=1033.130,21.891,410.053,168.574,41.812,157.815
C01531=1033.123,21.641,410.068,168.572,41.813,157.815
C01532=1033.117,21.392,410.084,168.570,41.814,157.815
C01533=1033.111,21.143,410.100,168.567,41.815,157.815
C01534=1033.105,20.893,410.115,168.565,41.816,157.815
C01535=1033.098,20.644,410.131,168.563,41.817,157.815
C01536=1033.092,20.395,410.147,168.560,41.818,157.815
C01537=1033.086,20.145,410.162,168.558,41.818,157.815
C01538=1033.079,19.896,410.178,168.555,41.819,157.815
C01539=1033.073,19.646,410.194,168.553,41.820,157.815
C01540=1033.067,19.397,410.209,168.551,41.820,157.815
C01541=1033.061,19.147,410.225,168.548,41.821,157.815
C01542=1033.055,18.898,410.240,168.547,41.822,157.815
C01543=1033.048,18.649,410.256,168.544,41.823,157.815
C01544=1033.042,18.399,410.272,168.542,41.824,157.816
C01545=1033.036,18.150,410.287,168.539,41.825,157.815
C01546=1033.029,17.900,410.303,168.537,41.826,157.815
C01547=1033.023,17.651,410.318,168.535,41.827,157.816
C01548=1033.016,17.401,410.334,168.532,41.828,157.816
C01549=1033.010,17.151,410.349,168.530,41.829,157.816
C01550=1033.004,16.902,410.366,168.527,41.829,157.816
C01551=1032.997,16.652,410.380,168.526,41.830,157.816
C01552=1032.991,16.403,410.396,168.524,41.831,157.816
C01553=1032.984,16.153,410.411,168.521,41.832,157.816
C01554=1032.978,15.904,410.427,168.519,41.832,157.816
C01555=1032.972,15.655,410.442,168.516,41.833,157.816
C01556=1032.966,15.406,410.458,168.514,41.834,157.816
C01557=1032.960,15.156,410.473,168.511,41.835,157.816
C01558=1032.953,14.907,410.489,168.509,41.836,157.816
C01559=1032.947,14.657,410.504,168.507,41.836,157.816
C01560=1032.941,14.408,410.520,168.504,41.838,157.816
C01561=1032.935,14.158,410.535,168.503,41.838,157.816
C01562=1032.928,13.909,410.550,168.500,41.839,157.816
C01563=1032.922,13.659,410.566,168.498,41.840,157.816
C01564=1032.916,13.410,410.581,168.495,41.841,157.816
C01565=1032.910,13.160,410.596,168.493,41.842,157.816
C01566=1032.903,12.911,410.612,168.490,41.843,157.816
C01567=1032.897,12.661,410.627,168.488,41.844,157.816
C01568=1032.889,12.376,410.644,168.485,41.845,157.816
C01569=1032.881,12.091,410.662,168.483,41.846,157.816
C01570=1032.875,11.806,410.679,168.480,41.847,157.816
C01571=1032.867,11.521,410.696,168.478,41.848,157.816
C01572=1032.860,11.272,410.711,168.475,41.849,157.816
C01573=1032.854,11.022,410.727,168.473,41.850,157.816
C01574=1032.848,10.772,410.742,168.470,41.851,157.816
C01575=1032.841,10.523,410.757,168.468,41.852,157.816
C01576=1032.835,10.274,410.772,168.465,41.852,157.816
C01577=1032.828,10.024,410.787,168.463,41.853,157.816
C01578=1032.822,9.774,410.802,168.461,41.854,157.816
C01579=1032.816,9.525,410.817,168.459,41.855,157.816
C01580=1032.810,9.276,410.833,168.456,41.856,157.816
C01581=1032.803,9.027,410.847,168.454,41.857,157.816
C01582=1032.797,8.777,410.862,168.451,41.858,157.816
C01583=1032.790,8.527,410.877,168.449,41.859,157.816
C01584=1032.784,8.278,410.892,168.446,41.860,157.816
C01585=1032.777,8.029,410.908,168.444,41.861,157.816
C01586=1032.771,7.779,410.923,168.442,41.862,157.816
C01587=1032.765,7.529,410.938,168.440,41.863,157.816
C01588=1032.759,7.280,410.952,168.437,41.864,157.816
C01589=1032.752,7.031,410.967,168.435,41.865,157.816
C01590=1032.746,6.781,410.982,168.432,41.866,157.816
C01591=1032.739,6.532,410.998,168.430,41.866,157.816
C01592=1032.733,6.282,411.013,168.427,41.867,157.816
C01593=1032.727,6.033,411.028,168.425,41.868,157.816
C01594=1032.720,5.783,411.043,168.422,41.869,157.816
C01595=1032.714,5.534,411.057,168.421,41.870,157.817
C01596=1032.708,5.284,411.072,168.418,41.871,157.817
C01597=1032.702,5.035,411.087,168.416,41.871,157.816
C01598=1032.695,4.785,411.102,168.413,41.873,157.816
C01599=1032.689,4.535,411.117,168.411,41.873,157.817
C01600=1032.682,4.286,411.133,168.408,41.875,157.817
C01601=1032.676,4.037,411.147,168.406,41.876,157.817
C01602=1032.670,3.788,411.162,168.403,41.877,157.817
C01603=1032.664,3.538,411.177,168.401,41.877,157.817
C01604=1032.657,3.288,411.192,168.399,41.878,157.817
C01605=1032.651,3.040,411.207,168.397,41.879,157.817
C01606=1032.645,2.790,411.222,168.395,41.880,157.817
C01607=1032.639,2.540,411.237,168.392,41.881,157.817
C01608=1032.632,2.291,411.252,168.390,41.881,157.817
C01609=1032.626,2.041,411.267,168.387,41.882,157.817
C01610=1032.620,1.792,411.281,168.385,41.883,157.817
C01611=1032.614,1.542,411.296,168.382,41.884,157.817
C01612=1032.607,1.293,411.311,168.380,41.885,157.817
C01613=1032.601,1.043,411.326,168.377,41.886,157.817
C01614=1032.595,0.794,411.341,168.376,41.887,157.817
C01615=1032.589,0.544,411.356,168.373,41.888,157.817
C01616=1032.582,0.295,411.371,168.371,41.889,157.817
C01617=1032.577,0.046,411.385,168.368,41.890,157.817
C01618=1032.570,-0.204,411.400,168.366,41.890,157.817
C01619=1032.564,-0.454,411.415,168.363,41.891,157.817
C01620=1032.557,-0.703,411.430,168.361,41.892,157.817
C01621=1032.552,-0.952,411.445,168.358,41.893,157.817
C01622=1032.546,-1.202,411.459,168.356,41.893,157.817
C01623=1032.539,-1.452,411.474,168.353,41.894,157.817
C01624=1032.533,-1.701,411.488,168.352,41.895,157.817
C01625=1032.527,-1.951,411.503,168.349,41.896,157.817
C01626=1032.521,-2.200,411.518,168.347,41.897,157.817
C01627=1032.515,-2.449,411.533,168.344,41.898,157.817
C01628=1032.509,-2.699,411.548,168.342,41.899,157.817
C01629=1032.502,-2.949,411.563,168.339,41.900,157.817
C01630=1032.496,-3.198,411.577,168.337,41.901,157.817
C01631=1032.490,-3.448,411.591,168.334,41.901,157.817
C01632=1032.484,-3.720,411.608,168.331,41.902,157.817
C01633=1032.477,-3.993,411.623,168.329,41.903,157.817
C01634=1032.469,-4.266,411.639,168.327,41.904,157.817
C01635=1032.463,-4.538,411.655,168.324,41.905,157.817
C01636=1032.456,-4.788,411.669,168.321,41.906,157.817
C01637=1032.450,-5.038,411.684,168.319,41.907,157.817
C01638=1032.444,-5.287,411.699,168.316,41.908,157.817
C01639=1032.437,-5.537,411.712,168.314,41.909,157.817
C01640=1032.430,-5.797,411.728,168.311,41.910,157.817
C01641=1032.423,-6.056,411.743,168.309,41.911,157.817
C01642=1032.417,-6.317,411.758,168.307,41.912,157.817
C01643=1032.411,-6.577,411.773,168.304,41.913,157.817
C01644=1032.404,-6.826,411.787,168.301,41.915,157.817
C01645=1032.398,-7.076,411.801,168.299,41.915,157.817
C01646=1032.392,-7.325,411.816,168.296,41.917,157.817
C01647=1032.385,-7.575,411.830,168.294,41.918,157.817
C01648=1032.379,-7.824,411.844,168.291,41.919,157.817
C01649=1032.372,-8.073,411.859,168.289,41.920,157.817
C01650=1032.367,-8.323,411.872,168.287,41.921,157.817
C01651=1032.360,-8.573,411.887,168.284,41.922,157.817
C01652=1032.353,-8.822,411.902,168.282,41.923,157.818
C01653=1032.348,-9.072,411.916,168.279,41.924,157.818
C01654=1032.341,-9.321,411.931,168.277,41.925,157.818
C01655=1032.335,-9.571,411.944,168.274,41.926,157.818
C01656=1032.329,-9.820,411.959,168.272,41.927,157.818
C01657=1032.322,-10.070,411.973,168.270,41.927,157.818
C01658=1032.316,-10.319,411.987,168.267,41.928,157.818
C01659=1032.310,-10.569,412.002,168.265,41.929,157.818
C01660=1032.303,-10.818,412.015,168.262,41.930,157.818
C01661=1032.297,-11.068,412.030,168.260,41.931,157.818
C01662=1032.291,-11.317,412.043,168.257,41.932,157.818
C01663=1032.284,-11.567,412.058,168.254,41.933,157.818
C01664=1032.279,-11.816,412.072,168.253,41.934,157.818
C01665=1032.272,-12.066,412.087,168.250,41.935,157.818
C01666=1032.266,-12.316,412.101,168.248,41.936,157.818
C01667=1032.259,-12.564,412.115,168.245,41.937,157.818
C01668=1032.253,-12.815,412.129,168.242,41.938,157.818
C01669=1032.247,-13.064,412.144,168.240,41.939,157.818
C01670=1032.241,-13.314,412.157,168.237,41.940,157.818
C01671=1032.235,-13.563,412.172,168.235,41.941,157.818
C01672=1032.228,-13.813,412.185,168.232,41.942,157.818
C01673=1032.223,-14.062,412.199,168.230,41.943,157.818
C01674=1032.216,-14.312,412.214,168.228,41.944,157.818
C01675=1032.210,-14.561,412.228,168.225,41.945,157.818
C01676=1032.204,-14.811,412.242,168.223,41.946,157.818
C01677=1032.197,-15.060,412.256,168.220,41.947,157.818
C01678=1032.191,-15.310,412.270,168.217,41.947,157.818
C01679=1032.185,-15.559,412.285,168.215,41.948,157.818
C01680=1032.179,-15.809,412.298,168.212,41.949,157.818
C01681=1032.172,-16.058,412.311,168.211,41.951,157.818
C01682=1032.166,-16.308,412.326,168.208,41.952,157.818
C01683=1032.160,-16.557,412.340,168.205,41.953,157.818
C01684=1032.153,-16.807,412.353,168.203,41.954,157.818
C01685=1032.148,-17.057,412.367,168.200,41.955,157.818
C01686=1032.140,-17.306,412.382,168.197,41.956,157.818
C01687=1032.134,-17.556,412.395,168.195,41.957,157.818
C01688=1032.128,-17.806,412.409,168.193,41.958,157.818
C01689=1032.122,-18.055,412.422,168.190,41.959,157.818
C01690=1032.115,-18.304,412.436,168.188,41.960,157.818
C01691=1032.109,-18.554,412.451,168.185,41.961,157.818
C01692=1032.103,-18.803,412.464,168.182,41.962,157.819
C01693=1032.096,-19.053,412.477,168.180,41.963,157.819
C01694=1032.091,-19.302,412.492,168.177,41.965,157.819
C01695=1032.084,-19.552,412.506,168.175,41.966,157.819
C01696=1032.077,-19.834,412.521,168.172,41.967,157.819
C01697=1032.070,-20.115,412.536,168.169,41.968,157.819
C01698=1032.063,-20.397,412.553,168.166,41.970,157.819
C01699=1032.055,-20.678,412.567,168.163,41.971,157.819
C01700=1032.050,-20.928,412.581,168.161,41.972,157.819
C01701=1032.043,-21.178,412.594,168.159,41.973,157.819
C01702=1032.036,-21.426,412.608,168.156,41.974,157.819
C01703=1032.030,-21.677,412.623,168.154,41.975,157.819
C01704=1032.024,-21.926,412.636,168.151,41.976,157.819
C01705=1032.018,-22.175,412.649,168.149,41.977,157.819
C01706=1032.012,-22.425,412.663,168.146,41.978,157.819
C01707=1032.006,-22.675,412.677,168.143,41.979,157.819
C01708=1031.999,-22.924,412.690,168.142,41.980,157.819
C01709=1031.993,-23.174,412.704,168.139,41.981,157.819
C01710=1031.987,-23.424,412.717,168.136,41.982,157.819
C01711=1031.981,-23.673,412.731,168.134,41.983,157.819
C01712=1031.974,-23.922,412.745,168.131,41.984,157.819
C01713=1031.968,-24.172,412.759,168.128,41.985,157.819
C01714=1031.962,-24.421,412.772,168.126,41.986,157.819
C01715=1031.955,-24.671,412.786,168.123,41.987,157.819
C01716=1031.950,-24.921,412.800,168.121,41.988,157.819
C01717=1031.944,-25.170,412.813,168.119,41.989,157.819
C01718=1031.937,-25.420,412.827,168.116,41.990,157.819
C01719=1031.931,-25.669,412.840,168.113,41.991,157.819
C01720=1031.925,-25.919,412.854,168.111,41.992,157.819
C01721=1031.918,-26.169,412.867,168.108,41.993,157.819
C01722=1031.912,-26.418,412.881,168.105,41.994,157.819
C01723=1031.907,-26.667,412.895,168.104,41.995,157.819
C01724=1031.900,-26.917,412.908,168.101,41.996,157.819
C01725=1031.894,-27.167,412.921,168.098,41.998,157.820
C01726=1031.888,-27.417,412.934,168.095,41.999,157.820
C01727=1031.881,-27.666,412.947,168.093,42.000,157.820
C01728=1031.875,-27.916,412.961,168.090,42.001,157.820
C01729=1031.868,-28.165,412.974,168.087,42.002,157.820
C01730=1031.862,-28.414,412.987,168.085,42.003,157.820
C01731=1031.856,-28.664,413.001,168.083,42.004,157.820
C01732=1031.849,-28.914,413.014,168.080,42.006,157.820
C01733=1031.843,-29.163,413.027,168.077,42.007,157.820
C01734=1031.837,-29.413,413.040,168.075,42.008,157.820
C01735=1031.831,-29.662,413.053,168.072,42.009,157.820
C01736=1031.825,-29.912,413.068,168.069,42.010,157.820
C01737=1031.819,-30.161,413.081,168.067,42.011,157.820
C01738=1031.813,-30.411,413.093,168.065,42.012,157.820
C01739=1031.806,-30.661,413.107,168.062,42.014,157.820
C01740=1031.800,-30.911,413.120,168.059,42.015,157.820
C01741=1031.793,-31.160,413.134,168.056,42.016,157.820
C01742=1031.788,-31.410,413.146,168.054,42.017,157.820
C01743=1031.781,-31.659,413.159,168.052,42.018,157.820
C01744=1031.775,-31.909,413.173,168.049,42.019,157.820
C01745=1031.768,-32.158,413.186,168.047,42.020,157.820
C01746=1031.762,-32.408,413.199,168.044,42.021,157.820
C01747=1031.756,-32.657,413.212,168.041,42.022,157.820
C01748=1031.750,-32.907,413.225,168.038,42.024,157.820
C01749=1031.743,-33.157,413.238,168.037,42.025,157.821
C01750=1031.737,-33.406,413.252,168.034,42.026,157.821
C01751=1031.731,-33.656,413.265,168.031,42.027,157.821
C01752=1031.725,-33.905,413.278,168.028,42.028,157.821
C01753=1031.719,-34.155,413.291,168.026,42.029,157.821
C01754=1031.713,-34.404,413.304,168.023,42.030,157.821
C01755=1031.707,-34.654,413.317,168.020,42.031,157.821
C01756=1031.700,-34.904,413.330,168.018,42.032,157.821
C01757=1031.694,-35.153,413.343,168.016,42.034,157.821
C01758=1031.688,-35.403,413.356,168.013,42.035,157.821
C01759=1031.682,-35.652,413.369,168.010,42.036,157.821
C01760=1031.675,-35.933,413.383,168.007,42.037,157.821
C01761=1031.667,-36.214,413.399,168.004,42.038,157.821
C01762=1031.660,-36.495,413.413,168.001,42.039,157.821
C01763=1031.653,-36.775,413.427,167.999,42.041,157.821
C01764=1031.647,-37.025,413.440,167.996,42.042,157.821
C01765=1031.641,-37.275,413.454,167.993,42.043,157.821
C01766=1031.635,-37.524,413.466,167.990,42.044,157.821
C01767=1031.629,-37.774,413.479,167.988,42.045,157.821
C01768=1031.622,-38.023,413.493,167.985,42.046,157.821
C01769=1031.616,-38.273,413.505,167.983,42.047,157.821
C01770=1031.610,-38.522,413.518,167.980,42.048,157.821
C01771=1031.604,-38.772,413.531,167.978,42.049,157.821
C01772=1031.598,-39.021,413.544,167.975,42.051,157.821
C01773=1031.592,-39.271,413.557,167.972,42.052,157.821
C01774=1031.586,-39.521,413.569,167.969,42.053,157.821
C01775=1031.579,-39.770,413.582,167.968,42.054,157.821
C01776=1031.573,-40.020,413.595,167.965,42.056,157.822
C01777=1031.567,-40.270,413.608,167.962,42.057,157.822
C01778=1031.560,-40.519,413.620,167.959,42.058,157.822
C01779=1031.554,-40.769,413.633,167.956,42.059,157.822
C01780=1031.548,-41.019,413.646,167.954,42.061,157.822
C01781=1031.542,-41.268,413.659,167.952,42.062,157.822
C01782=1031.535,-41.517,413.671,167.949,42.063,157.822
C01783=1031.529,-41.767,413.684,167.946,42.064,157.822
C01784=1031.523,-42.017,413.696,167.943,42.066,157.822
C01785=1031.516,-42.266,413.709,167.940,42.067,157.822
C01786=1031.510,-42.516,413.722,167.939,42.068,157.822
C01787=1031.504,-42.766,413.734,167.936,42.069,157.822
C01788=1031.498,-43.015,413.747,167.933,42.070,157.822
C01789=1031.491,-43.265,413.759,167.930,42.072,157.822
C01790=1031.486,-43.515,413.772,167.927,42.073,157.822
C01791=1031.480,-43.764,413.785,167.924,42.074,157.822
C01792=1031.473,-44.013,413.797,167.923,42.075,157.822
C01793=1031.467,-44.263,413.810,167.920,42.077,157.822
C01794=1031.461,-44.513,413.822,167.917,42.078,157.822
C01795=1031.454,-44.762,413.835,167.914,42.079,157.822
C01796=1031.448,-45.012,413.848,167.911,42.080,157.822
C01797=1031.442,-45.262,413.860,167.910,42.082,157.823
C01798=1031.436,-45.512,413.873,167.907,42.083,157.823
C01799=1031.429,-45.761,413.885,167.904,42.084,157.823
C01800=1031.423,-46.011,413.898,167.901,42.085,157.823
C01801=1031.417,-46.261,413.910,167.898,42.086,157.823
C01802=1031.411,-46.509,413.922,167.895,42.088,157.823
C01803=1031.406,-46.759,413.935,167.894,42.089,157.823
C01804=1031.399,-47.009,413.948,167.891,42.090,157.823
C01805=1031.393,-47.258,413.960,167.888,42.091,157.823
C01806=1031.387,-47.508,413.972,167.885,42.093,157.823
C01807=1031.381,-47.758,413.985,167.882,42.094,157.823
C01808=1031.374,-48.007,413.997,167.879,42.095,157.823
C01809=1031.368,-48.257,414.009,167.878,42.096,157.823
C01810=1031.362,-48.507,414.022,167.875,42.097,157.823
C01811=1031.355,-48.756,414.035,167.872,42.099,157.823
C01812=1031.350,-49.005,414.047,167.869,42.100,157.823
C01813=1031.344,-49.255,414.059,167.866,42.101,157.823
C01814=1031.338,-49.505,414.071,167.863,42.102,157.823
C01815=1031.332,-49.755,414.084,167.862,42.103,157.823
C01816=1031.326,-50.005,414.096,167.859,42.105,157.823
C01817=1031.319,-50.254,414.108,167.856,42.106,157.823
C01818=1031.313,-50.504,414.121,167.853,42.107,157.823
